// TIA Portal V18 export
// export: Created 2026-06-23T08:49:30.0253939Z, ExportSetting WithDefaults, DisplayName Totally Integrated Automation Portal, DisplayVersion V18, DisplayName TIA Portal Openness, DisplayVersion V18, DisplayName TIA Portal Version Control Interface, DisplayVersion V18, DisplayName STEP 7 Professional, DisplayVersion V18, DisplayName STEP 7 Safety, DisplayVersion V18, DisplayName WinCC Professional, DisplayVersion V18
FUNCTION "FC_Manual_Control_PLC1" : Void   // FC62, LAD
{ S7_Optimized_Access := 'TRUE' }
VERSION : 0.1
// stored: AutoNumber true, IsIECCheckEnabled false, SetENOAutomatically false, UDAEnableTagReadback false
BEGIN

REGION Network 1: Xác định trạng thái Manual Mode Active PLC1
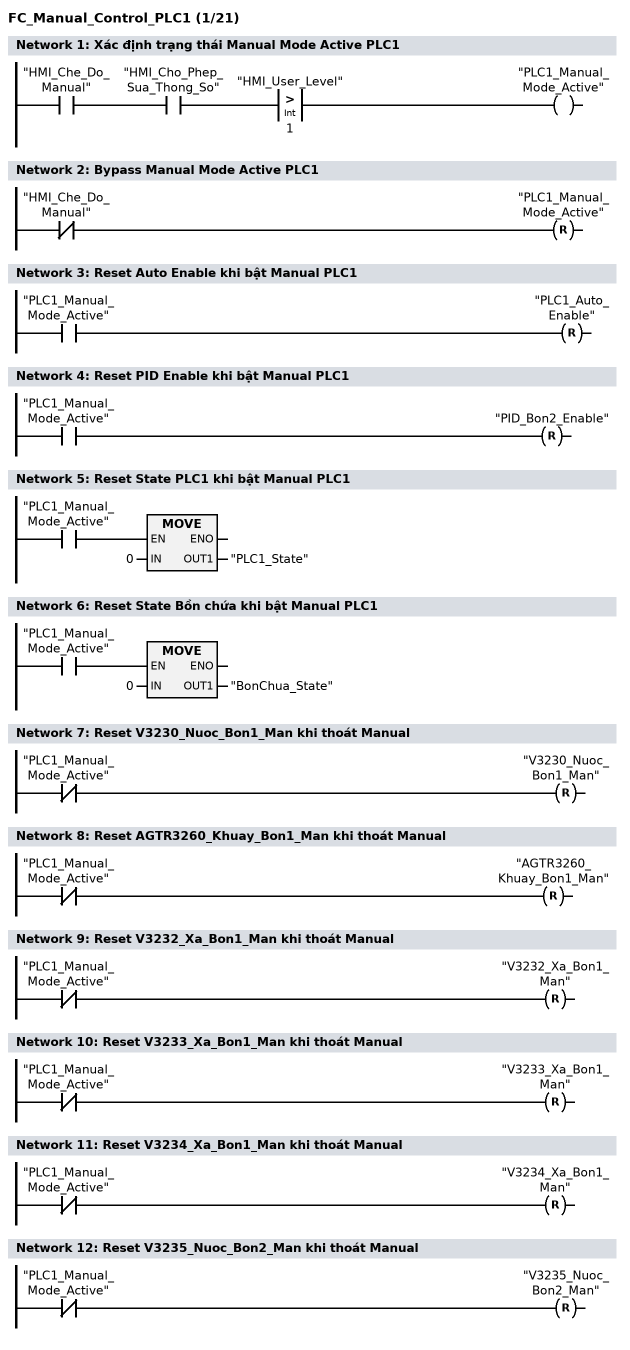
   RUNG wire#powerrail
      Contact( "HMI_Che_Do_Manual" )
      Contact( "HMI_Cho_Phep_Sua_Thong_So" )
      { S7_Templates := "SrcType := Int" } GT_Contact(in1 := "HMI_User_Level", in2 := 1)
      Coil( "PLC1_Manual_Mode_Active" )
   END_RUNG
   // the same network as SCL:
   "PLC1_Manual_Mode_Active" := "HMI_Che_Do_Manual" AND "HMI_Cho_Phep_Sua_Thong_So" AND ("HMI_User_Level" > 1);
END_REGION

REGION Network 2: Bypass Manual Mode Active PLC1
   RUNG wire#powerrail
      I_Contact( "HMI_Che_Do_Manual" )
      R_Coil( "PLC1_Manual_Mode_Active" )
   END_RUNG
   // the same network as SCL:
   IF NOT "HMI_Che_Do_Manual" THEN "PLC1_Manual_Mode_Active" := FALSE; END_IF;
END_REGION

REGION Network 3: Reset Auto Enable khi bật Manual PLC1
   RUNG wire#powerrail
      Contact( "PLC1_Manual_Mode_Active" )
      R_Coil( "PLC1_Auto_Enable" )
   END_RUNG
   // the same network as SCL:
   IF "PLC1_Manual_Mode_Active" THEN "PLC1_Auto_Enable" := FALSE; END_IF;
END_REGION

REGION Network 4: Reset PID Enable khi bật Manual PLC1
   RUNG wire#powerrail
      Contact( "PLC1_Manual_Mode_Active" )
      R_Coil( "PID_Bon2_Enable" )
   END_RUNG
   // the same network as SCL:
   IF "PLC1_Manual_Mode_Active" THEN "PID_Bon2_Enable" := FALSE; END_IF;
END_REGION

REGION Network 5: Reset State PLC1 khi bật Manual PLC1
   RUNG wire#powerrail
      Contact( "PLC1_Manual_Mode_Active" )
      { S7_GenerateENO := "TRUE" } Move(in := 0, out1 => "PLC1_State")
   END_RUNG
   // the same network as SCL:
   IF "PLC1_Manual_Mode_Active" THEN "PLC1_State" := 0; END_IF;
END_REGION

REGION Network 6: Reset State Bồn chứa khi bật Manual PLC1
   RUNG wire#powerrail
      Contact( "PLC1_Manual_Mode_Active" )
      { S7_GenerateENO := "TRUE" } Move(in := 0, out1 => "BonChua_State")
   END_RUNG
   // the same network as SCL:
   IF "PLC1_Manual_Mode_Active" THEN "BonChua_State" := 0; END_IF;
END_REGION

REGION Network 7: Reset V3230_Nuoc_Bon1_Man khi thoát Manual
   RUNG wire#powerrail
      I_Contact( "PLC1_Manual_Mode_Active" )
      R_Coil( "V3230_Nuoc_Bon1_Man" )
   END_RUNG
   // the same network as SCL:
   IF NOT "PLC1_Manual_Mode_Active" THEN "V3230_Nuoc_Bon1_Man" := FALSE; END_IF;
END_REGION

REGION Network 8: Reset AGTR3260_Khuay_Bon1_Man khi thoát Manual
   RUNG wire#powerrail
      I_Contact( "PLC1_Manual_Mode_Active" )
      R_Coil( "AGTR3260_Khuay_Bon1_Man" )
   END_RUNG
   // the same network as SCL:
   IF NOT "PLC1_Manual_Mode_Active" THEN "AGTR3260_Khuay_Bon1_Man" := FALSE; END_IF;
END_REGION

REGION Network 9: Reset V3232_Xa_Bon1_Man khi thoát Manual
   RUNG wire#powerrail
      I_Contact( "PLC1_Manual_Mode_Active" )
      R_Coil( "V3232_Xa_Bon1_Man" )
   END_RUNG
   // the same network as SCL:
   IF NOT "PLC1_Manual_Mode_Active" THEN "V3232_Xa_Bon1_Man" := FALSE; END_IF;
END_REGION

REGION Network 10: Reset V3233_Xa_Bon1_Man khi thoát Manual
   RUNG wire#powerrail
      I_Contact( "PLC1_Manual_Mode_Active" )
      R_Coil( "V3233_Xa_Bon1_Man" )
   END_RUNG
   // the same network as SCL:
   IF NOT "PLC1_Manual_Mode_Active" THEN "V3233_Xa_Bon1_Man" := FALSE; END_IF;
END_REGION

REGION Network 11: Reset V3234_Xa_Bon1_Man khi thoát Manual
   RUNG wire#powerrail
      I_Contact( "PLC1_Manual_Mode_Active" )
      R_Coil( "V3234_Xa_Bon1_Man" )
   END_RUNG
   // the same network as SCL:
   IF NOT "PLC1_Manual_Mode_Active" THEN "V3234_Xa_Bon1_Man" := FALSE; END_IF;
END_REGION

REGION Network 12: Reset V3235_Nuoc_Bon2_Man khi thoát Manual
   RUNG wire#powerrail
      I_Contact( "PLC1_Manual_Mode_Active" )
      R_Coil( "V3235_Nuoc_Bon2_Man" )
   END_RUNG
   // the same network as SCL:
   IF NOT "PLC1_Manual_Mode_Active" THEN "V3235_Nuoc_Bon2_Man" := FALSE; END_IF;
END_REGION

REGION Network 13: Reset VFD_Bon2_Run_Man khi thoát Manual
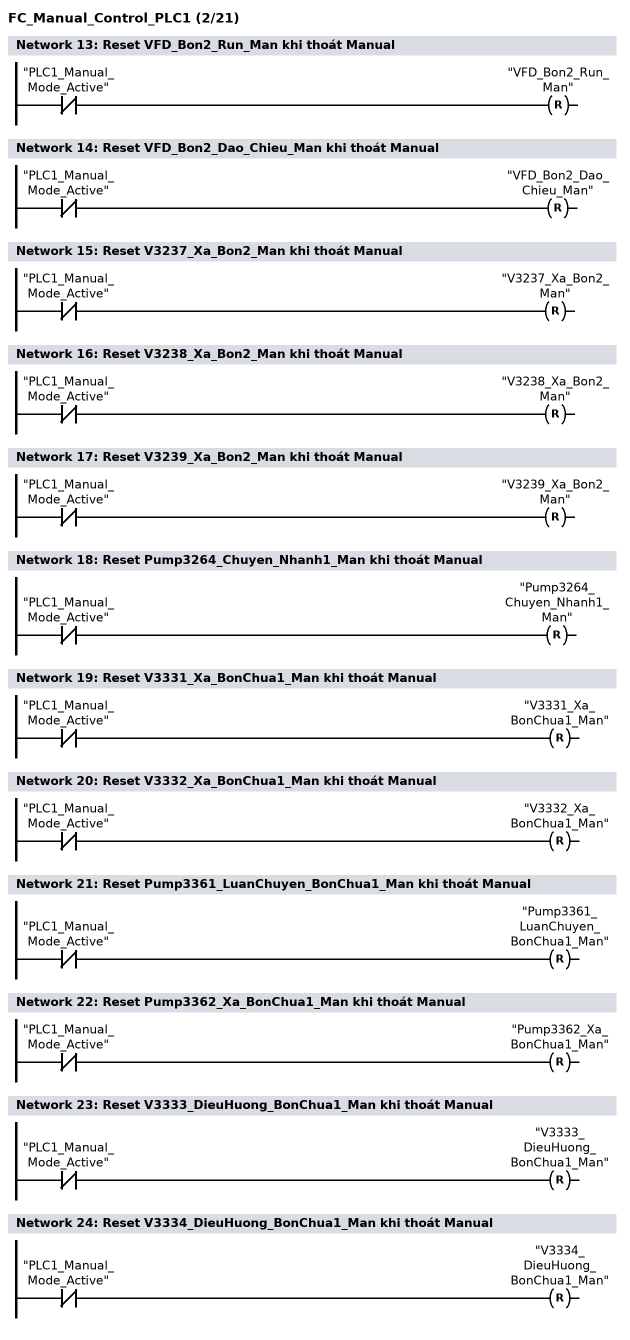
   RUNG wire#powerrail
      I_Contact( "PLC1_Manual_Mode_Active" )
      R_Coil( "VFD_Bon2_Run_Man" )
   END_RUNG
   // the same network as SCL:
   IF NOT "PLC1_Manual_Mode_Active" THEN "VFD_Bon2_Run_Man" := FALSE; END_IF;
END_REGION

REGION Network 14: Reset VFD_Bon2_Dao_Chieu_Man khi thoát Manual
   RUNG wire#powerrail
      I_Contact( "PLC1_Manual_Mode_Active" )
      R_Coil( "VFD_Bon2_Dao_Chieu_Man" )
   END_RUNG
   // the same network as SCL:
   IF NOT "PLC1_Manual_Mode_Active" THEN "VFD_Bon2_Dao_Chieu_Man" := FALSE; END_IF;
END_REGION

REGION Network 15: Reset V3237_Xa_Bon2_Man khi thoát Manual
   RUNG wire#powerrail
      I_Contact( "PLC1_Manual_Mode_Active" )
      R_Coil( "V3237_Xa_Bon2_Man" )
   END_RUNG
   // the same network as SCL:
   IF NOT "PLC1_Manual_Mode_Active" THEN "V3237_Xa_Bon2_Man" := FALSE; END_IF;
END_REGION

REGION Network 16: Reset V3238_Xa_Bon2_Man khi thoát Manual
   RUNG wire#powerrail
      I_Contact( "PLC1_Manual_Mode_Active" )
      R_Coil( "V3238_Xa_Bon2_Man" )
   END_RUNG
   // the same network as SCL:
   IF NOT "PLC1_Manual_Mode_Active" THEN "V3238_Xa_Bon2_Man" := FALSE; END_IF;
END_REGION

REGION Network 17: Reset V3239_Xa_Bon2_Man khi thoát Manual
   RUNG wire#powerrail
      I_Contact( "PLC1_Manual_Mode_Active" )
      R_Coil( "V3239_Xa_Bon2_Man" )
   END_RUNG
   // the same network as SCL:
   IF NOT "PLC1_Manual_Mode_Active" THEN "V3239_Xa_Bon2_Man" := FALSE; END_IF;
END_REGION

REGION Network 18: Reset Pump3264_Chuyen_Nhanh1_Man khi thoát Manual
   RUNG wire#powerrail
      I_Contact( "PLC1_Manual_Mode_Active" )
      R_Coil( "Pump3264_Chuyen_Nhanh1_Man" )
   END_RUNG
   // the same network as SCL:
   IF NOT "PLC1_Manual_Mode_Active" THEN "Pump3264_Chuyen_Nhanh1_Man" := FALSE; END_IF;
END_REGION

REGION Network 19: Reset V3331_Xa_BonChua1_Man khi thoát Manual
   RUNG wire#powerrail
      I_Contact( "PLC1_Manual_Mode_Active" )
      R_Coil( "V3331_Xa_BonChua1_Man" )
   END_RUNG
   // the same network as SCL:
   IF NOT "PLC1_Manual_Mode_Active" THEN "V3331_Xa_BonChua1_Man" := FALSE; END_IF;
END_REGION

REGION Network 20: Reset V3332_Xa_BonChua1_Man khi thoát Manual
   RUNG wire#powerrail
      I_Contact( "PLC1_Manual_Mode_Active" )
      R_Coil( "V3332_Xa_BonChua1_Man" )
   END_RUNG
   // the same network as SCL:
   IF NOT "PLC1_Manual_Mode_Active" THEN "V3332_Xa_BonChua1_Man" := FALSE; END_IF;
END_REGION

REGION Network 21: Reset Pump3361_LuanChuyen_BonChua1_Man khi thoát Manual
   RUNG wire#powerrail
      I_Contact( "PLC1_Manual_Mode_Active" )
      R_Coil( "Pump3361_LuanChuyen_BonChua1_Man" )
   END_RUNG
   // the same network as SCL:
   IF NOT "PLC1_Manual_Mode_Active" THEN "Pump3361_LuanChuyen_BonChua1_Man" := FALSE; END_IF;
END_REGION

REGION Network 22: Reset Pump3362_Xa_BonChua1_Man khi thoát Manual
   RUNG wire#powerrail
      I_Contact( "PLC1_Manual_Mode_Active" )
      R_Coil( "Pump3362_Xa_BonChua1_Man" )
   END_RUNG
   // the same network as SCL:
   IF NOT "PLC1_Manual_Mode_Active" THEN "Pump3362_Xa_BonChua1_Man" := FALSE; END_IF;
END_REGION

REGION Network 23: Reset V3333_DieuHuong_BonChua1_Man khi thoát Manual
   RUNG wire#powerrail
      I_Contact( "PLC1_Manual_Mode_Active" )
      R_Coil( "V3333_DieuHuong_BonChua1_Man" )
   END_RUNG
   // the same network as SCL:
   IF NOT "PLC1_Manual_Mode_Active" THEN "V3333_DieuHuong_BonChua1_Man" := FALSE; END_IF;
END_REGION

REGION Network 24: Reset V3334_DieuHuong_BonChua1_Man khi thoát Manual
   RUNG wire#powerrail
      I_Contact( "PLC1_Manual_Mode_Active" )
      R_Coil( "V3334_DieuHuong_BonChua1_Man" )
   END_RUNG
   // the same network as SCL:
   IF NOT "PLC1_Manual_Mode_Active" THEN "V3334_DieuHuong_BonChua1_Man" := FALSE; END_IF;
END_REGION

REGION Network 25: Reset V3335_DieuHuong_BonChua1_Man khi thoát Manual
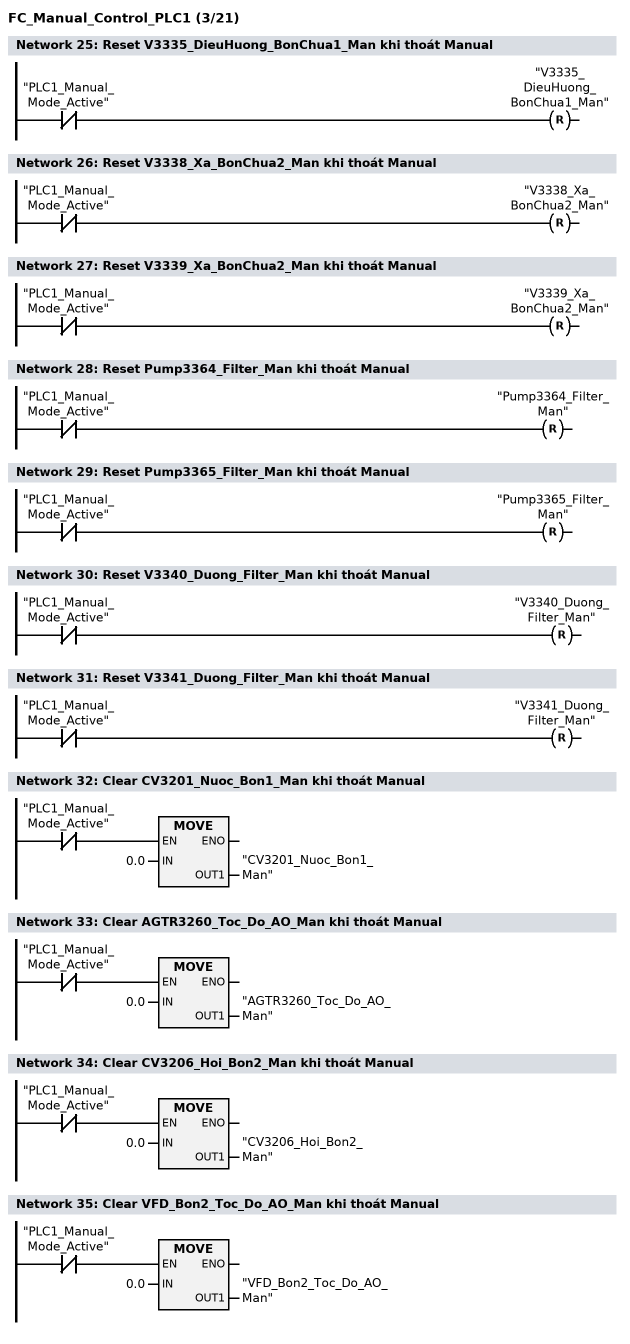
   RUNG wire#powerrail
      I_Contact( "PLC1_Manual_Mode_Active" )
      R_Coil( "V3335_DieuHuong_BonChua1_Man" )
   END_RUNG
   // the same network as SCL:
   IF NOT "PLC1_Manual_Mode_Active" THEN "V3335_DieuHuong_BonChua1_Man" := FALSE; END_IF;
END_REGION

REGION Network 26: Reset V3338_Xa_BonChua2_Man khi thoát Manual
   RUNG wire#powerrail
      I_Contact( "PLC1_Manual_Mode_Active" )
      R_Coil( "V3338_Xa_BonChua2_Man" )
   END_RUNG
   // the same network as SCL:
   IF NOT "PLC1_Manual_Mode_Active" THEN "V3338_Xa_BonChua2_Man" := FALSE; END_IF;
END_REGION

REGION Network 27: Reset V3339_Xa_BonChua2_Man khi thoát Manual
   RUNG wire#powerrail
      I_Contact( "PLC1_Manual_Mode_Active" )
      R_Coil( "V3339_Xa_BonChua2_Man" )
   END_RUNG
   // the same network as SCL:
   IF NOT "PLC1_Manual_Mode_Active" THEN "V3339_Xa_BonChua2_Man" := FALSE; END_IF;
END_REGION

REGION Network 28: Reset Pump3364_Filter_Man khi thoát Manual
   RUNG wire#powerrail
      I_Contact( "PLC1_Manual_Mode_Active" )
      R_Coil( "Pump3364_Filter_Man" )
   END_RUNG
   // the same network as SCL:
   IF NOT "PLC1_Manual_Mode_Active" THEN "Pump3364_Filter_Man" := FALSE; END_IF;
END_REGION

REGION Network 29: Reset Pump3365_Filter_Man khi thoát Manual
   RUNG wire#powerrail
      I_Contact( "PLC1_Manual_Mode_Active" )
      R_Coil( "Pump3365_Filter_Man" )
   END_RUNG
   // the same network as SCL:
   IF NOT "PLC1_Manual_Mode_Active" THEN "Pump3365_Filter_Man" := FALSE; END_IF;
END_REGION

REGION Network 30: Reset V3340_Duong_Filter_Man khi thoát Manual
   RUNG wire#powerrail
      I_Contact( "PLC1_Manual_Mode_Active" )
      R_Coil( "V3340_Duong_Filter_Man" )
   END_RUNG
   // the same network as SCL:
   IF NOT "PLC1_Manual_Mode_Active" THEN "V3340_Duong_Filter_Man" := FALSE; END_IF;
END_REGION

REGION Network 31: Reset V3341_Duong_Filter_Man khi thoát Manual
   RUNG wire#powerrail
      I_Contact( "PLC1_Manual_Mode_Active" )
      R_Coil( "V3341_Duong_Filter_Man" )
   END_RUNG
   // the same network as SCL:
   IF NOT "PLC1_Manual_Mode_Active" THEN "V3341_Duong_Filter_Man" := FALSE; END_IF;
END_REGION

REGION Network 32: Clear CV3201_Nuoc_Bon1_Man khi thoát Manual
   RUNG wire#powerrail
      I_Contact( "PLC1_Manual_Mode_Active" )
      { S7_GenerateENO := "TRUE" } Move(in := 0.0, out1 => "CV3201_Nuoc_Bon1_Man")
   END_RUNG
   // the same network as SCL:
   IF NOT "PLC1_Manual_Mode_Active" THEN "CV3201_Nuoc_Bon1_Man" := 0.0; END_IF;
END_REGION

REGION Network 33: Clear AGTR3260_Toc_Do_AO_Man khi thoát Manual
   RUNG wire#powerrail
      I_Contact( "PLC1_Manual_Mode_Active" )
      { S7_GenerateENO := "TRUE" } Move(in := 0.0, out1 => "AGTR3260_Toc_Do_AO_Man")
   END_RUNG
   // the same network as SCL:
   IF NOT "PLC1_Manual_Mode_Active" THEN "AGTR3260_Toc_Do_AO_Man" := 0.0; END_IF;
END_REGION

REGION Network 34: Clear CV3206_Hoi_Bon2_Man khi thoát Manual
   RUNG wire#powerrail
      I_Contact( "PLC1_Manual_Mode_Active" )
      { S7_GenerateENO := "TRUE" } Move(in := 0.0, out1 => "CV3206_Hoi_Bon2_Man")
   END_RUNG
   // the same network as SCL:
   IF NOT "PLC1_Manual_Mode_Active" THEN "CV3206_Hoi_Bon2_Man" := 0.0; END_IF;
END_REGION

REGION Network 35: Clear VFD_Bon2_Toc_Do_AO_Man khi thoát Manual
   RUNG wire#powerrail
      I_Contact( "PLC1_Manual_Mode_Active" )
      { S7_GenerateENO := "TRUE" } Move(in := 0.0, out1 => "VFD_Bon2_Toc_Do_AO_Man")
   END_RUNG
   // the same network as SCL:
   IF NOT "PLC1_Manual_Mode_Active" THEN "VFD_Bon2_Toc_Do_AO_Man" := 0.0; END_IF;
END_REGION

REGION Network 36: Clear CV3304_Nuoc_Lam_Mat_Man khi thoát Manual
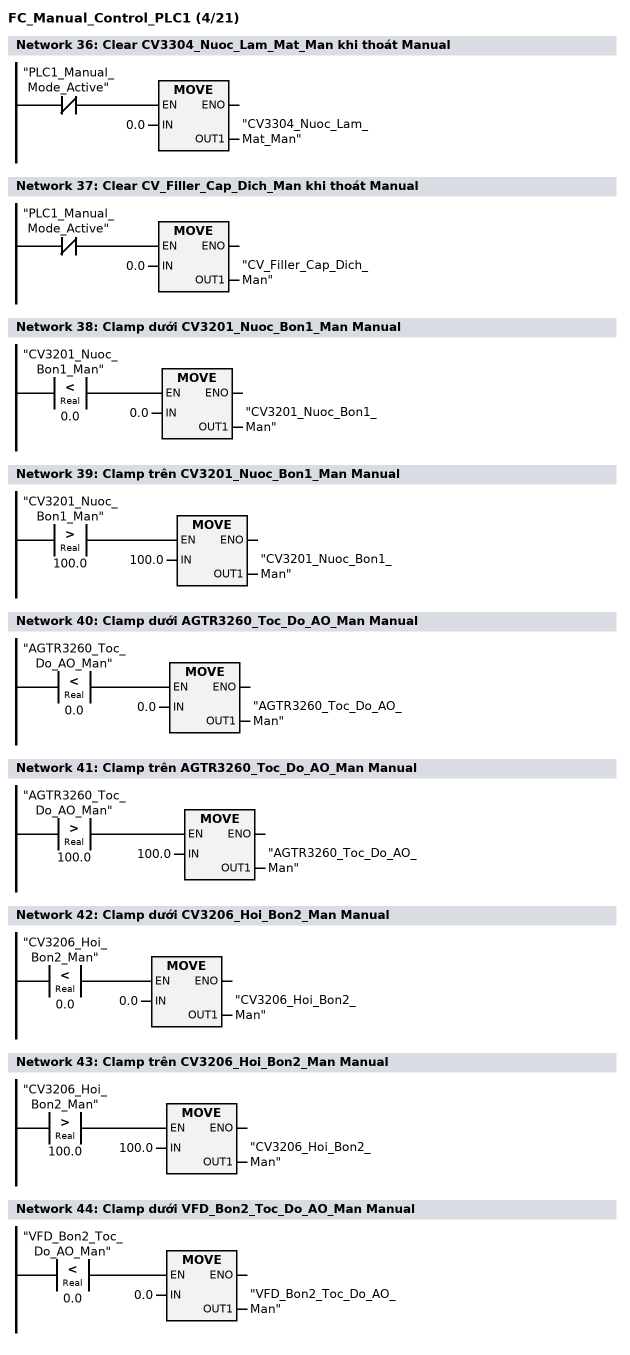
   RUNG wire#powerrail
      I_Contact( "PLC1_Manual_Mode_Active" )
      { S7_GenerateENO := "TRUE" } Move(in := 0.0, out1 => "CV3304_Nuoc_Lam_Mat_Man")
   END_RUNG
   // the same network as SCL:
   IF NOT "PLC1_Manual_Mode_Active" THEN "CV3304_Nuoc_Lam_Mat_Man" := 0.0; END_IF;
END_REGION

REGION Network 37: Clear CV_Filler_Cap_Dich_Man khi thoát Manual
   RUNG wire#powerrail
      I_Contact( "PLC1_Manual_Mode_Active" )
      { S7_GenerateENO := "TRUE" } Move(in := 0.0, out1 => "CV_Filler_Cap_Dich_Man")
   END_RUNG
   // the same network as SCL:
   IF NOT "PLC1_Manual_Mode_Active" THEN "CV_Filler_Cap_Dich_Man" := 0.0; END_IF;
END_REGION

REGION Network 38: Clamp dưới CV3201_Nuoc_Bon1_Man Manual
   RUNG wire#powerrail
      { S7_Templates := "SrcType := Real" } LT_Contact(in1 := "CV3201_Nuoc_Bon1_Man", in2 := 0.0)
      { S7_GenerateENO := "TRUE" } Move(in := 0.0, out1 => "CV3201_Nuoc_Bon1_Man")
   END_RUNG
   // the same network as SCL:
   IF "CV3201_Nuoc_Bon1_Man" < 0.0 THEN "CV3201_Nuoc_Bon1_Man" := 0.0; END_IF;
END_REGION

REGION Network 39: Clamp trên CV3201_Nuoc_Bon1_Man Manual
   RUNG wire#powerrail
      { S7_Templates := "SrcType := Real" } GT_Contact(in1 := "CV3201_Nuoc_Bon1_Man", in2 := 100.0)
      { S7_GenerateENO := "TRUE" } Move(in := 100.0, out1 => "CV3201_Nuoc_Bon1_Man")
   END_RUNG
   // the same network as SCL:
   IF "CV3201_Nuoc_Bon1_Man" > 100.0 THEN "CV3201_Nuoc_Bon1_Man" := 100.0; END_IF;
END_REGION

REGION Network 40: Clamp dưới AGTR3260_Toc_Do_AO_Man Manual
   RUNG wire#powerrail
      { S7_Templates := "SrcType := Real" } LT_Contact(in1 := "AGTR3260_Toc_Do_AO_Man", in2 := 0.0)
      { S7_GenerateENO := "TRUE" } Move(in := 0.0, out1 => "AGTR3260_Toc_Do_AO_Man")
   END_RUNG
   // the same network as SCL:
   IF "AGTR3260_Toc_Do_AO_Man" < 0.0 THEN "AGTR3260_Toc_Do_AO_Man" := 0.0; END_IF;
END_REGION

REGION Network 41: Clamp trên AGTR3260_Toc_Do_AO_Man Manual
   RUNG wire#powerrail
      { S7_Templates := "SrcType := Real" } GT_Contact(in1 := "AGTR3260_Toc_Do_AO_Man", in2 := 100.0)
      { S7_GenerateENO := "TRUE" } Move(in := 100.0, out1 => "AGTR3260_Toc_Do_AO_Man")
   END_RUNG
   // the same network as SCL:
   IF "AGTR3260_Toc_Do_AO_Man" > 100.0 THEN "AGTR3260_Toc_Do_AO_Man" := 100.0; END_IF;
END_REGION

REGION Network 42: Clamp dưới CV3206_Hoi_Bon2_Man Manual
   RUNG wire#powerrail
      { S7_Templates := "SrcType := Real" } LT_Contact(in1 := "CV3206_Hoi_Bon2_Man", in2 := 0.0)
      { S7_GenerateENO := "TRUE" } Move(in := 0.0, out1 => "CV3206_Hoi_Bon2_Man")
   END_RUNG
   // the same network as SCL:
   IF "CV3206_Hoi_Bon2_Man" < 0.0 THEN "CV3206_Hoi_Bon2_Man" := 0.0; END_IF;
END_REGION

REGION Network 43: Clamp trên CV3206_Hoi_Bon2_Man Manual
   RUNG wire#powerrail
      { S7_Templates := "SrcType := Real" } GT_Contact(in1 := "CV3206_Hoi_Bon2_Man", in2 := 100.0)
      { S7_GenerateENO := "TRUE" } Move(in := 100.0, out1 => "CV3206_Hoi_Bon2_Man")
   END_RUNG
   // the same network as SCL:
   IF "CV3206_Hoi_Bon2_Man" > 100.0 THEN "CV3206_Hoi_Bon2_Man" := 100.0; END_IF;
END_REGION

REGION Network 44: Clamp dưới VFD_Bon2_Toc_Do_AO_Man Manual
   RUNG wire#powerrail
      { S7_Templates := "SrcType := Real" } LT_Contact(in1 := "VFD_Bon2_Toc_Do_AO_Man", in2 := 0.0)
      { S7_GenerateENO := "TRUE" } Move(in := 0.0, out1 => "VFD_Bon2_Toc_Do_AO_Man")
   END_RUNG
   // the same network as SCL:
   IF "VFD_Bon2_Toc_Do_AO_Man" < 0.0 THEN "VFD_Bon2_Toc_Do_AO_Man" := 0.0; END_IF;
END_REGION

REGION Network 45: Clamp trên VFD_Bon2_Toc_Do_AO_Man Manual
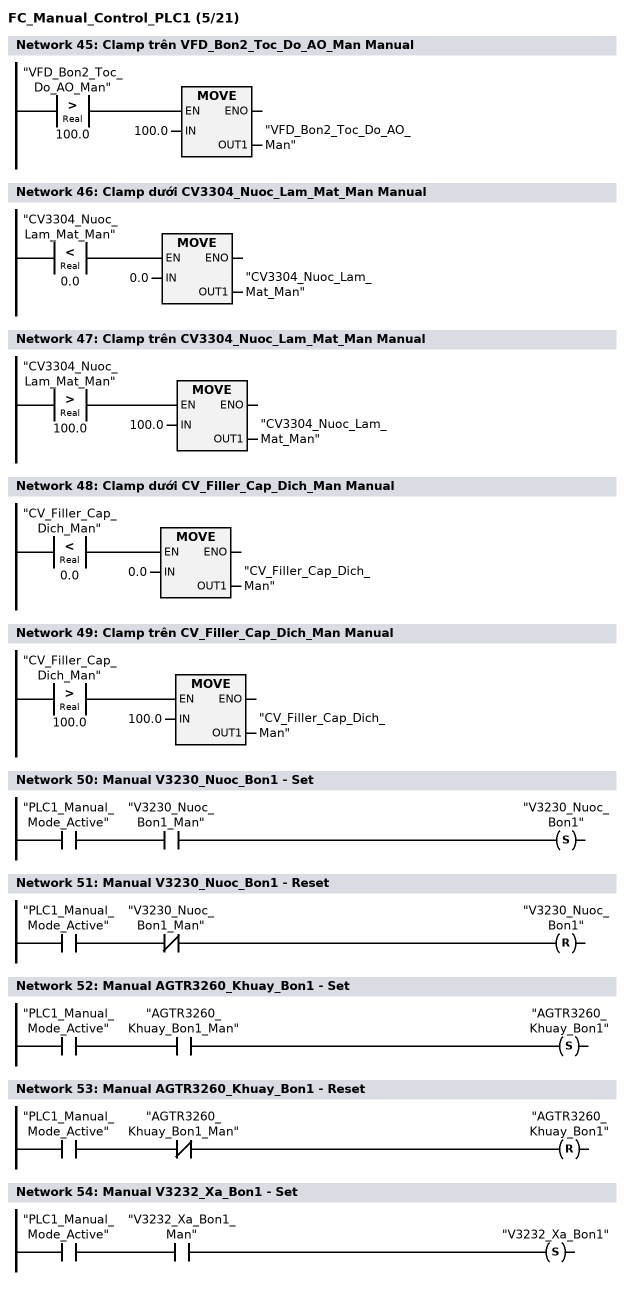
   RUNG wire#powerrail
      { S7_Templates := "SrcType := Real" } GT_Contact(in1 := "VFD_Bon2_Toc_Do_AO_Man", in2 := 100.0)
      { S7_GenerateENO := "TRUE" } Move(in := 100.0, out1 => "VFD_Bon2_Toc_Do_AO_Man")
   END_RUNG
   // the same network as SCL:
   IF "VFD_Bon2_Toc_Do_AO_Man" > 100.0 THEN "VFD_Bon2_Toc_Do_AO_Man" := 100.0; END_IF;
END_REGION

REGION Network 46: Clamp dưới CV3304_Nuoc_Lam_Mat_Man Manual
   RUNG wire#powerrail
      { S7_Templates := "SrcType := Real" } LT_Contact(in1 := "CV3304_Nuoc_Lam_Mat_Man", in2 := 0.0)
      { S7_GenerateENO := "TRUE" } Move(in := 0.0, out1 => "CV3304_Nuoc_Lam_Mat_Man")
   END_RUNG
   // the same network as SCL:
   IF "CV3304_Nuoc_Lam_Mat_Man" < 0.0 THEN "CV3304_Nuoc_Lam_Mat_Man" := 0.0; END_IF;
END_REGION

REGION Network 47: Clamp trên CV3304_Nuoc_Lam_Mat_Man Manual
   RUNG wire#powerrail
      { S7_Templates := "SrcType := Real" } GT_Contact(in1 := "CV3304_Nuoc_Lam_Mat_Man", in2 := 100.0)
      { S7_GenerateENO := "TRUE" } Move(in := 100.0, out1 => "CV3304_Nuoc_Lam_Mat_Man")
   END_RUNG
   // the same network as SCL:
   IF "CV3304_Nuoc_Lam_Mat_Man" > 100.0 THEN "CV3304_Nuoc_Lam_Mat_Man" := 100.0; END_IF;
END_REGION

REGION Network 48: Clamp dưới CV_Filler_Cap_Dich_Man Manual
   RUNG wire#powerrail
      { S7_Templates := "SrcType := Real" } LT_Contact(in1 := "CV_Filler_Cap_Dich_Man", in2 := 0.0)
      { S7_GenerateENO := "TRUE" } Move(in := 0.0, out1 => "CV_Filler_Cap_Dich_Man")
   END_RUNG
   // the same network as SCL:
   IF "CV_Filler_Cap_Dich_Man" < 0.0 THEN "CV_Filler_Cap_Dich_Man" := 0.0; END_IF;
END_REGION

REGION Network 49: Clamp trên CV_Filler_Cap_Dich_Man Manual
   RUNG wire#powerrail
      { S7_Templates := "SrcType := Real" } GT_Contact(in1 := "CV_Filler_Cap_Dich_Man", in2 := 100.0)
      { S7_GenerateENO := "TRUE" } Move(in := 100.0, out1 => "CV_Filler_Cap_Dich_Man")
   END_RUNG
   // the same network as SCL:
   IF "CV_Filler_Cap_Dich_Man" > 100.0 THEN "CV_Filler_Cap_Dich_Man" := 100.0; END_IF;
END_REGION

REGION Network 50: Manual V3230_Nuoc_Bon1 - Set
   RUNG wire#powerrail
      Contact( "PLC1_Manual_Mode_Active" )
      Contact( "V3230_Nuoc_Bon1_Man" )
      S_Coil( "V3230_Nuoc_Bon1" )
   END_RUNG
   // the same network as SCL:
   IF "PLC1_Manual_Mode_Active" AND "V3230_Nuoc_Bon1_Man" THEN "V3230_Nuoc_Bon1" := TRUE; END_IF;
END_REGION

REGION Network 51: Manual V3230_Nuoc_Bon1 - Reset
   RUNG wire#powerrail
      Contact( "PLC1_Manual_Mode_Active" )
      I_Contact( "V3230_Nuoc_Bon1_Man" )
      R_Coil( "V3230_Nuoc_Bon1" )
   END_RUNG
   // the same network as SCL:
   IF "PLC1_Manual_Mode_Active" AND NOT "V3230_Nuoc_Bon1_Man" THEN "V3230_Nuoc_Bon1" := FALSE; END_IF;
END_REGION

REGION Network 52: Manual AGTR3260_Khuay_Bon1 - Set
   RUNG wire#powerrail
      Contact( "PLC1_Manual_Mode_Active" )
      Contact( "AGTR3260_Khuay_Bon1_Man" )
      S_Coil( "AGTR3260_Khuay_Bon1" )
   END_RUNG
   // the same network as SCL:
   IF "PLC1_Manual_Mode_Active" AND "AGTR3260_Khuay_Bon1_Man" THEN "AGTR3260_Khuay_Bon1" := TRUE; END_IF;
END_REGION

REGION Network 53: Manual AGTR3260_Khuay_Bon1 - Reset
   RUNG wire#powerrail
      Contact( "PLC1_Manual_Mode_Active" )
      I_Contact( "AGTR3260_Khuay_Bon1_Man" )
      R_Coil( "AGTR3260_Khuay_Bon1" )
   END_RUNG
   // the same network as SCL:
   IF "PLC1_Manual_Mode_Active" AND NOT "AGTR3260_Khuay_Bon1_Man" THEN
       "AGTR3260_Khuay_Bon1" := FALSE;
   END_IF;
END_REGION

REGION Network 54: Manual V3232_Xa_Bon1 - Set
   RUNG wire#powerrail
      Contact( "PLC1_Manual_Mode_Active" )
      Contact( "V3232_Xa_Bon1_Man" )
      S_Coil( "V3232_Xa_Bon1" )
   END_RUNG
   // the same network as SCL:
   IF "PLC1_Manual_Mode_Active" AND "V3232_Xa_Bon1_Man" THEN "V3232_Xa_Bon1" := TRUE; END_IF;
END_REGION

REGION Network 55: Manual V3232_Xa_Bon1 - Reset
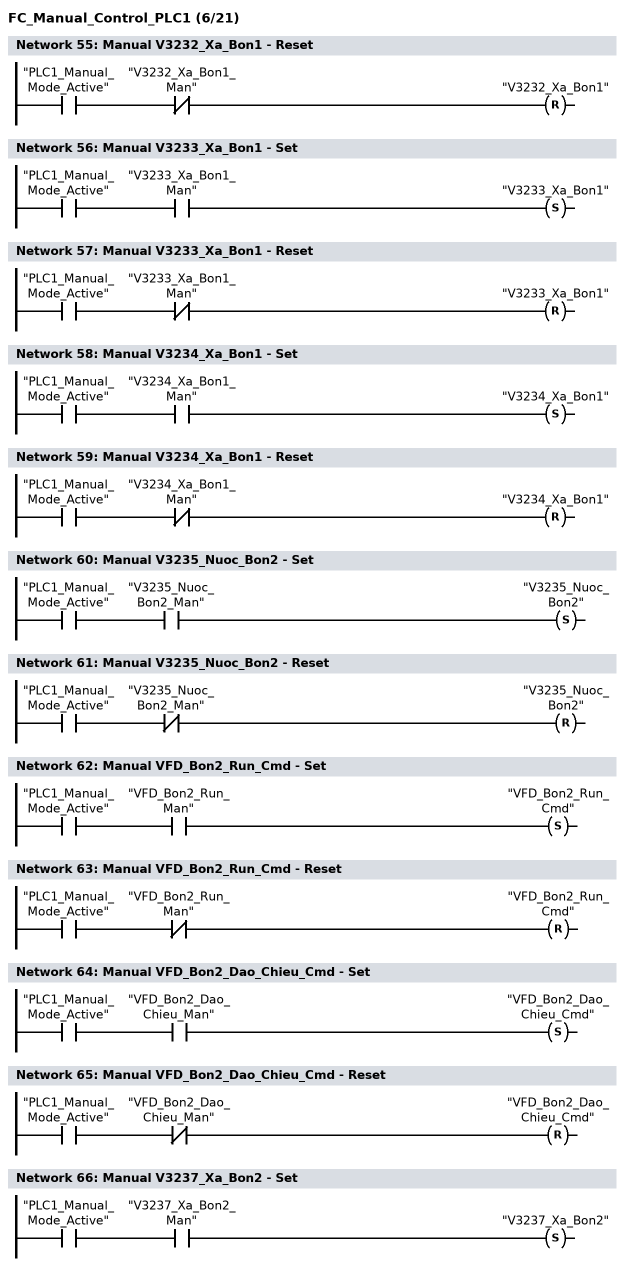
   RUNG wire#powerrail
      Contact( "PLC1_Manual_Mode_Active" )
      I_Contact( "V3232_Xa_Bon1_Man" )
      R_Coil( "V3232_Xa_Bon1" )
   END_RUNG
   // the same network as SCL:
   IF "PLC1_Manual_Mode_Active" AND NOT "V3232_Xa_Bon1_Man" THEN "V3232_Xa_Bon1" := FALSE; END_IF;
END_REGION

REGION Network 56: Manual V3233_Xa_Bon1 - Set
   RUNG wire#powerrail
      Contact( "PLC1_Manual_Mode_Active" )
      Contact( "V3233_Xa_Bon1_Man" )
      S_Coil( "V3233_Xa_Bon1" )
   END_RUNG
   // the same network as SCL:
   IF "PLC1_Manual_Mode_Active" AND "V3233_Xa_Bon1_Man" THEN "V3233_Xa_Bon1" := TRUE; END_IF;
END_REGION

REGION Network 57: Manual V3233_Xa_Bon1 - Reset
   RUNG wire#powerrail
      Contact( "PLC1_Manual_Mode_Active" )
      I_Contact( "V3233_Xa_Bon1_Man" )
      R_Coil( "V3233_Xa_Bon1" )
   END_RUNG
   // the same network as SCL:
   IF "PLC1_Manual_Mode_Active" AND NOT "V3233_Xa_Bon1_Man" THEN "V3233_Xa_Bon1" := FALSE; END_IF;
END_REGION

REGION Network 58: Manual V3234_Xa_Bon1 - Set
   RUNG wire#powerrail
      Contact( "PLC1_Manual_Mode_Active" )
      Contact( "V3234_Xa_Bon1_Man" )
      S_Coil( "V3234_Xa_Bon1" )
   END_RUNG
   // the same network as SCL:
   IF "PLC1_Manual_Mode_Active" AND "V3234_Xa_Bon1_Man" THEN "V3234_Xa_Bon1" := TRUE; END_IF;
END_REGION

REGION Network 59: Manual V3234_Xa_Bon1 - Reset
   RUNG wire#powerrail
      Contact( "PLC1_Manual_Mode_Active" )
      I_Contact( "V3234_Xa_Bon1_Man" )
      R_Coil( "V3234_Xa_Bon1" )
   END_RUNG
   // the same network as SCL:
   IF "PLC1_Manual_Mode_Active" AND NOT "V3234_Xa_Bon1_Man" THEN "V3234_Xa_Bon1" := FALSE; END_IF;
END_REGION

REGION Network 60: Manual V3235_Nuoc_Bon2 - Set
   RUNG wire#powerrail
      Contact( "PLC1_Manual_Mode_Active" )
      Contact( "V3235_Nuoc_Bon2_Man" )
      S_Coil( "V3235_Nuoc_Bon2" )
   END_RUNG
   // the same network as SCL:
   IF "PLC1_Manual_Mode_Active" AND "V3235_Nuoc_Bon2_Man" THEN "V3235_Nuoc_Bon2" := TRUE; END_IF;
END_REGION

REGION Network 61: Manual V3235_Nuoc_Bon2 - Reset
   RUNG wire#powerrail
      Contact( "PLC1_Manual_Mode_Active" )
      I_Contact( "V3235_Nuoc_Bon2_Man" )
      R_Coil( "V3235_Nuoc_Bon2" )
   END_RUNG
   // the same network as SCL:
   IF "PLC1_Manual_Mode_Active" AND NOT "V3235_Nuoc_Bon2_Man" THEN "V3235_Nuoc_Bon2" := FALSE; END_IF;
END_REGION

REGION Network 62: Manual VFD_Bon2_Run_Cmd - Set
   RUNG wire#powerrail
      Contact( "PLC1_Manual_Mode_Active" )
      Contact( "VFD_Bon2_Run_Man" )
      S_Coil( "VFD_Bon2_Run_Cmd" )
   END_RUNG
   // the same network as SCL:
   IF "PLC1_Manual_Mode_Active" AND "VFD_Bon2_Run_Man" THEN "VFD_Bon2_Run_Cmd" := TRUE; END_IF;
END_REGION

REGION Network 63: Manual VFD_Bon2_Run_Cmd - Reset
   RUNG wire#powerrail
      Contact( "PLC1_Manual_Mode_Active" )
      I_Contact( "VFD_Bon2_Run_Man" )
      R_Coil( "VFD_Bon2_Run_Cmd" )
   END_RUNG
   // the same network as SCL:
   IF "PLC1_Manual_Mode_Active" AND NOT "VFD_Bon2_Run_Man" THEN "VFD_Bon2_Run_Cmd" := FALSE; END_IF;
END_REGION

REGION Network 64: Manual VFD_Bon2_Dao_Chieu_Cmd - Set
   RUNG wire#powerrail
      Contact( "PLC1_Manual_Mode_Active" )
      Contact( "VFD_Bon2_Dao_Chieu_Man" )
      S_Coil( "VFD_Bon2_Dao_Chieu_Cmd" )
   END_RUNG
   // the same network as SCL:
   IF "PLC1_Manual_Mode_Active" AND "VFD_Bon2_Dao_Chieu_Man" THEN "VFD_Bon2_Dao_Chieu_Cmd" := TRUE; END_IF;
END_REGION

REGION Network 65: Manual VFD_Bon2_Dao_Chieu_Cmd - Reset
   RUNG wire#powerrail
      Contact( "PLC1_Manual_Mode_Active" )
      I_Contact( "VFD_Bon2_Dao_Chieu_Man" )
      R_Coil( "VFD_Bon2_Dao_Chieu_Cmd" )
   END_RUNG
   // the same network as SCL:
   IF "PLC1_Manual_Mode_Active" AND NOT "VFD_Bon2_Dao_Chieu_Man" THEN
       "VFD_Bon2_Dao_Chieu_Cmd" := FALSE;
   END_IF;
END_REGION

REGION Network 66: Manual V3237_Xa_Bon2 - Set
   RUNG wire#powerrail
      Contact( "PLC1_Manual_Mode_Active" )
      Contact( "V3237_Xa_Bon2_Man" )
      S_Coil( "V3237_Xa_Bon2" )
   END_RUNG
   // the same network as SCL:
   IF "PLC1_Manual_Mode_Active" AND "V3237_Xa_Bon2_Man" THEN "V3237_Xa_Bon2" := TRUE; END_IF;
END_REGION

REGION Network 67: Manual V3237_Xa_Bon2 - Reset
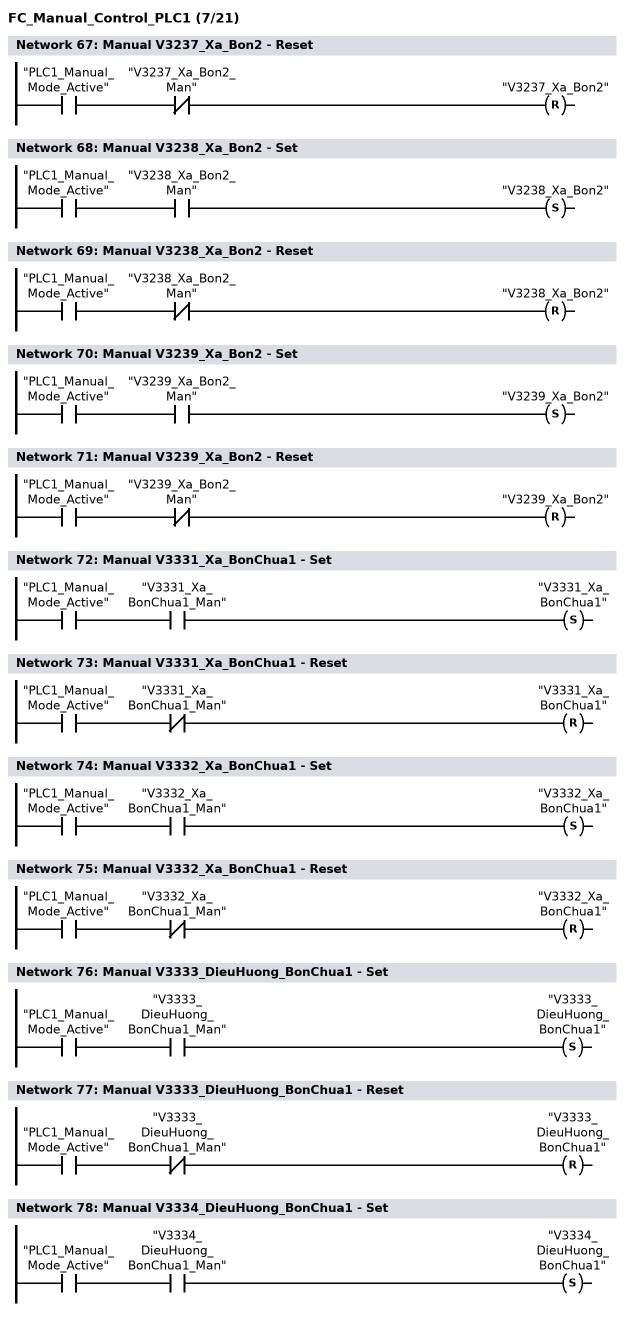
   RUNG wire#powerrail
      Contact( "PLC1_Manual_Mode_Active" )
      I_Contact( "V3237_Xa_Bon2_Man" )
      R_Coil( "V3237_Xa_Bon2" )
   END_RUNG
   // the same network as SCL:
   IF "PLC1_Manual_Mode_Active" AND NOT "V3237_Xa_Bon2_Man" THEN "V3237_Xa_Bon2" := FALSE; END_IF;
END_REGION

REGION Network 68: Manual V3238_Xa_Bon2 - Set
   RUNG wire#powerrail
      Contact( "PLC1_Manual_Mode_Active" )
      Contact( "V3238_Xa_Bon2_Man" )
      S_Coil( "V3238_Xa_Bon2" )
   END_RUNG
   // the same network as SCL:
   IF "PLC1_Manual_Mode_Active" AND "V3238_Xa_Bon2_Man" THEN "V3238_Xa_Bon2" := TRUE; END_IF;
END_REGION

REGION Network 69: Manual V3238_Xa_Bon2 - Reset
   RUNG wire#powerrail
      Contact( "PLC1_Manual_Mode_Active" )
      I_Contact( "V3238_Xa_Bon2_Man" )
      R_Coil( "V3238_Xa_Bon2" )
   END_RUNG
   // the same network as SCL:
   IF "PLC1_Manual_Mode_Active" AND NOT "V3238_Xa_Bon2_Man" THEN "V3238_Xa_Bon2" := FALSE; END_IF;
END_REGION

REGION Network 70: Manual V3239_Xa_Bon2 - Set
   RUNG wire#powerrail
      Contact( "PLC1_Manual_Mode_Active" )
      Contact( "V3239_Xa_Bon2_Man" )
      S_Coil( "V3239_Xa_Bon2" )
   END_RUNG
   // the same network as SCL:
   IF "PLC1_Manual_Mode_Active" AND "V3239_Xa_Bon2_Man" THEN "V3239_Xa_Bon2" := TRUE; END_IF;
END_REGION

REGION Network 71: Manual V3239_Xa_Bon2 - Reset
   RUNG wire#powerrail
      Contact( "PLC1_Manual_Mode_Active" )
      I_Contact( "V3239_Xa_Bon2_Man" )
      R_Coil( "V3239_Xa_Bon2" )
   END_RUNG
   // the same network as SCL:
   IF "PLC1_Manual_Mode_Active" AND NOT "V3239_Xa_Bon2_Man" THEN "V3239_Xa_Bon2" := FALSE; END_IF;
END_REGION

REGION Network 72: Manual V3331_Xa_BonChua1 - Set
   RUNG wire#powerrail
      Contact( "PLC1_Manual_Mode_Active" )
      Contact( "V3331_Xa_BonChua1_Man" )
      S_Coil( "V3331_Xa_BonChua1" )
   END_RUNG
   // the same network as SCL:
   IF "PLC1_Manual_Mode_Active" AND "V3331_Xa_BonChua1_Man" THEN "V3331_Xa_BonChua1" := TRUE; END_IF;
END_REGION

REGION Network 73: Manual V3331_Xa_BonChua1 - Reset
   RUNG wire#powerrail
      Contact( "PLC1_Manual_Mode_Active" )
      I_Contact( "V3331_Xa_BonChua1_Man" )
      R_Coil( "V3331_Xa_BonChua1" )
   END_RUNG
   // the same network as SCL:
   IF "PLC1_Manual_Mode_Active" AND NOT "V3331_Xa_BonChua1_Man" THEN "V3331_Xa_BonChua1" := FALSE; END_IF;
END_REGION

REGION Network 74: Manual V3332_Xa_BonChua1 - Set
   RUNG wire#powerrail
      Contact( "PLC1_Manual_Mode_Active" )
      Contact( "V3332_Xa_BonChua1_Man" )
      S_Coil( "V3332_Xa_BonChua1" )
   END_RUNG
   // the same network as SCL:
   IF "PLC1_Manual_Mode_Active" AND "V3332_Xa_BonChua1_Man" THEN "V3332_Xa_BonChua1" := TRUE; END_IF;
END_REGION

REGION Network 75: Manual V3332_Xa_BonChua1 - Reset
   RUNG wire#powerrail
      Contact( "PLC1_Manual_Mode_Active" )
      I_Contact( "V3332_Xa_BonChua1_Man" )
      R_Coil( "V3332_Xa_BonChua1" )
   END_RUNG
   // the same network as SCL:
   IF "PLC1_Manual_Mode_Active" AND NOT "V3332_Xa_BonChua1_Man" THEN "V3332_Xa_BonChua1" := FALSE; END_IF;
END_REGION

REGION Network 76: Manual V3333_DieuHuong_BonChua1 - Set
   RUNG wire#powerrail
      Contact( "PLC1_Manual_Mode_Active" )
      Contact( "V3333_DieuHuong_BonChua1_Man" )
      S_Coil( "V3333_DieuHuong_BonChua1" )
   END_RUNG
   // the same network as SCL:
   IF "PLC1_Manual_Mode_Active" AND "V3333_DieuHuong_BonChua1_Man" THEN
       "V3333_DieuHuong_BonChua1" := TRUE;
   END_IF;
END_REGION

REGION Network 77: Manual V3333_DieuHuong_BonChua1 - Reset
   RUNG wire#powerrail
      Contact( "PLC1_Manual_Mode_Active" )
      I_Contact( "V3333_DieuHuong_BonChua1_Man" )
      R_Coil( "V3333_DieuHuong_BonChua1" )
   END_RUNG
   // the same network as SCL:
   IF "PLC1_Manual_Mode_Active" AND NOT "V3333_DieuHuong_BonChua1_Man" THEN
       "V3333_DieuHuong_BonChua1" := FALSE;
   END_IF;
END_REGION

REGION Network 78: Manual V3334_DieuHuong_BonChua1 - Set
   RUNG wire#powerrail
      Contact( "PLC1_Manual_Mode_Active" )
      Contact( "V3334_DieuHuong_BonChua1_Man" )
      S_Coil( "V3334_DieuHuong_BonChua1" )
   END_RUNG
   // the same network as SCL:
   IF "PLC1_Manual_Mode_Active" AND "V3334_DieuHuong_BonChua1_Man" THEN
       "V3334_DieuHuong_BonChua1" := TRUE;
   END_IF;
END_REGION

REGION Network 79: Manual V3334_DieuHuong_BonChua1 - Reset
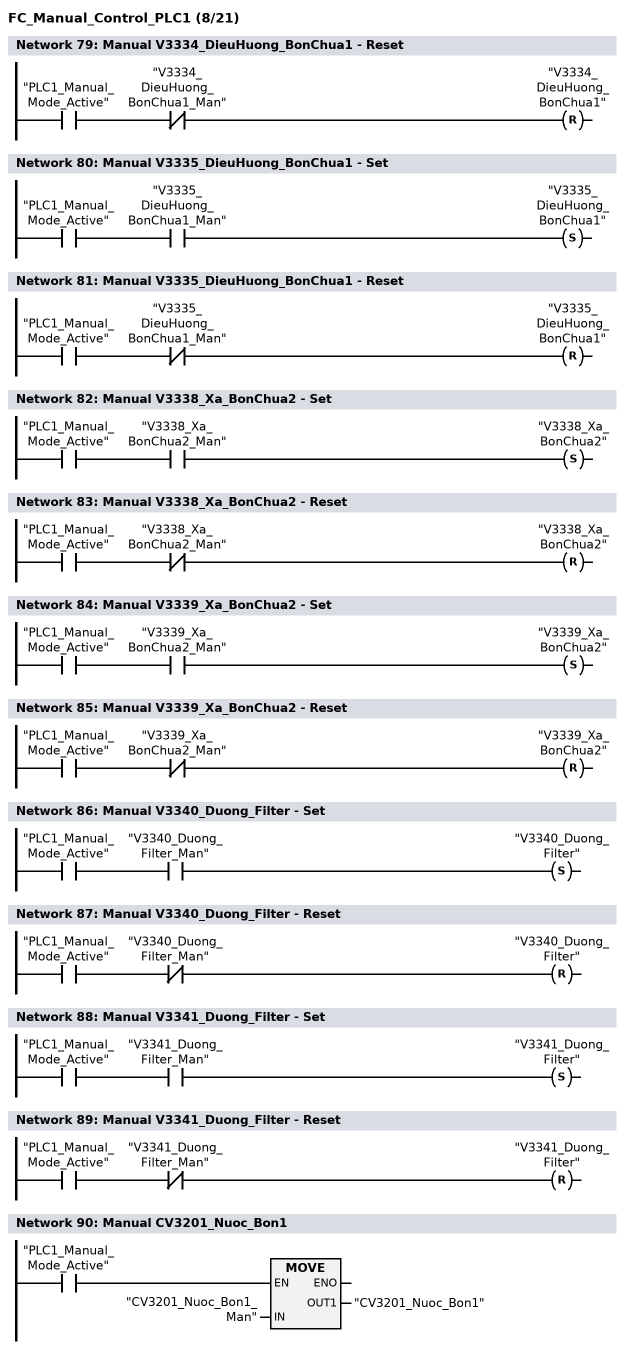
   RUNG wire#powerrail
      Contact( "PLC1_Manual_Mode_Active" )
      I_Contact( "V3334_DieuHuong_BonChua1_Man" )
      R_Coil( "V3334_DieuHuong_BonChua1" )
   END_RUNG
   // the same network as SCL:
   IF "PLC1_Manual_Mode_Active" AND NOT "V3334_DieuHuong_BonChua1_Man" THEN
       "V3334_DieuHuong_BonChua1" := FALSE;
   END_IF;
END_REGION

REGION Network 80: Manual V3335_DieuHuong_BonChua1 - Set
   RUNG wire#powerrail
      Contact( "PLC1_Manual_Mode_Active" )
      Contact( "V3335_DieuHuong_BonChua1_Man" )
      S_Coil( "V3335_DieuHuong_BonChua1" )
   END_RUNG
   // the same network as SCL:
   IF "PLC1_Manual_Mode_Active" AND "V3335_DieuHuong_BonChua1_Man" THEN
       "V3335_DieuHuong_BonChua1" := TRUE;
   END_IF;
END_REGION

REGION Network 81: Manual V3335_DieuHuong_BonChua1 - Reset
   RUNG wire#powerrail
      Contact( "PLC1_Manual_Mode_Active" )
      I_Contact( "V3335_DieuHuong_BonChua1_Man" )
      R_Coil( "V3335_DieuHuong_BonChua1" )
   END_RUNG
   // the same network as SCL:
   IF "PLC1_Manual_Mode_Active" AND NOT "V3335_DieuHuong_BonChua1_Man" THEN
       "V3335_DieuHuong_BonChua1" := FALSE;
   END_IF;
END_REGION

REGION Network 82: Manual V3338_Xa_BonChua2 - Set
   RUNG wire#powerrail
      Contact( "PLC1_Manual_Mode_Active" )
      Contact( "V3338_Xa_BonChua2_Man" )
      S_Coil( "V3338_Xa_BonChua2" )
   END_RUNG
   // the same network as SCL:
   IF "PLC1_Manual_Mode_Active" AND "V3338_Xa_BonChua2_Man" THEN "V3338_Xa_BonChua2" := TRUE; END_IF;
END_REGION

REGION Network 83: Manual V3338_Xa_BonChua2 - Reset
   RUNG wire#powerrail
      Contact( "PLC1_Manual_Mode_Active" )
      I_Contact( "V3338_Xa_BonChua2_Man" )
      R_Coil( "V3338_Xa_BonChua2" )
   END_RUNG
   // the same network as SCL:
   IF "PLC1_Manual_Mode_Active" AND NOT "V3338_Xa_BonChua2_Man" THEN "V3338_Xa_BonChua2" := FALSE; END_IF;
END_REGION

REGION Network 84: Manual V3339_Xa_BonChua2 - Set
   RUNG wire#powerrail
      Contact( "PLC1_Manual_Mode_Active" )
      Contact( "V3339_Xa_BonChua2_Man" )
      S_Coil( "V3339_Xa_BonChua2" )
   END_RUNG
   // the same network as SCL:
   IF "PLC1_Manual_Mode_Active" AND "V3339_Xa_BonChua2_Man" THEN "V3339_Xa_BonChua2" := TRUE; END_IF;
END_REGION

REGION Network 85: Manual V3339_Xa_BonChua2 - Reset
   RUNG wire#powerrail
      Contact( "PLC1_Manual_Mode_Active" )
      I_Contact( "V3339_Xa_BonChua2_Man" )
      R_Coil( "V3339_Xa_BonChua2" )
   END_RUNG
   // the same network as SCL:
   IF "PLC1_Manual_Mode_Active" AND NOT "V3339_Xa_BonChua2_Man" THEN "V3339_Xa_BonChua2" := FALSE; END_IF;
END_REGION

REGION Network 86: Manual V3340_Duong_Filter - Set
   RUNG wire#powerrail
      Contact( "PLC1_Manual_Mode_Active" )
      Contact( "V3340_Duong_Filter_Man" )
      S_Coil( "V3340_Duong_Filter" )
   END_RUNG
   // the same network as SCL:
   IF "PLC1_Manual_Mode_Active" AND "V3340_Duong_Filter_Man" THEN "V3340_Duong_Filter" := TRUE; END_IF;
END_REGION

REGION Network 87: Manual V3340_Duong_Filter - Reset
   RUNG wire#powerrail
      Contact( "PLC1_Manual_Mode_Active" )
      I_Contact( "V3340_Duong_Filter_Man" )
      R_Coil( "V3340_Duong_Filter" )
   END_RUNG
   // the same network as SCL:
   IF "PLC1_Manual_Mode_Active" AND NOT "V3340_Duong_Filter_Man" THEN "V3340_Duong_Filter" := FALSE; END_IF;
END_REGION

REGION Network 88: Manual V3341_Duong_Filter - Set
   RUNG wire#powerrail
      Contact( "PLC1_Manual_Mode_Active" )
      Contact( "V3341_Duong_Filter_Man" )
      S_Coil( "V3341_Duong_Filter" )
   END_RUNG
   // the same network as SCL:
   IF "PLC1_Manual_Mode_Active" AND "V3341_Duong_Filter_Man" THEN "V3341_Duong_Filter" := TRUE; END_IF;
END_REGION

REGION Network 89: Manual V3341_Duong_Filter - Reset
   RUNG wire#powerrail
      Contact( "PLC1_Manual_Mode_Active" )
      I_Contact( "V3341_Duong_Filter_Man" )
      R_Coil( "V3341_Duong_Filter" )
   END_RUNG
   // the same network as SCL:
   IF "PLC1_Manual_Mode_Active" AND NOT "V3341_Duong_Filter_Man" THEN "V3341_Duong_Filter" := FALSE; END_IF;
END_REGION

REGION Network 90: Manual CV3201_Nuoc_Bon1
   RUNG wire#powerrail
      Contact( "PLC1_Manual_Mode_Active" )
      { S7_GenerateENO := "TRUE" } Move(in := "CV3201_Nuoc_Bon1_Man", out1 => "CV3201_Nuoc_Bon1")
   END_RUNG
   // the same network as SCL:
   IF "PLC1_Manual_Mode_Active" THEN "CV3201_Nuoc_Bon1" := "CV3201_Nuoc_Bon1_Man"; END_IF;
END_REGION

REGION Network 91: Manual AGTR3260_Toc_Do_AO
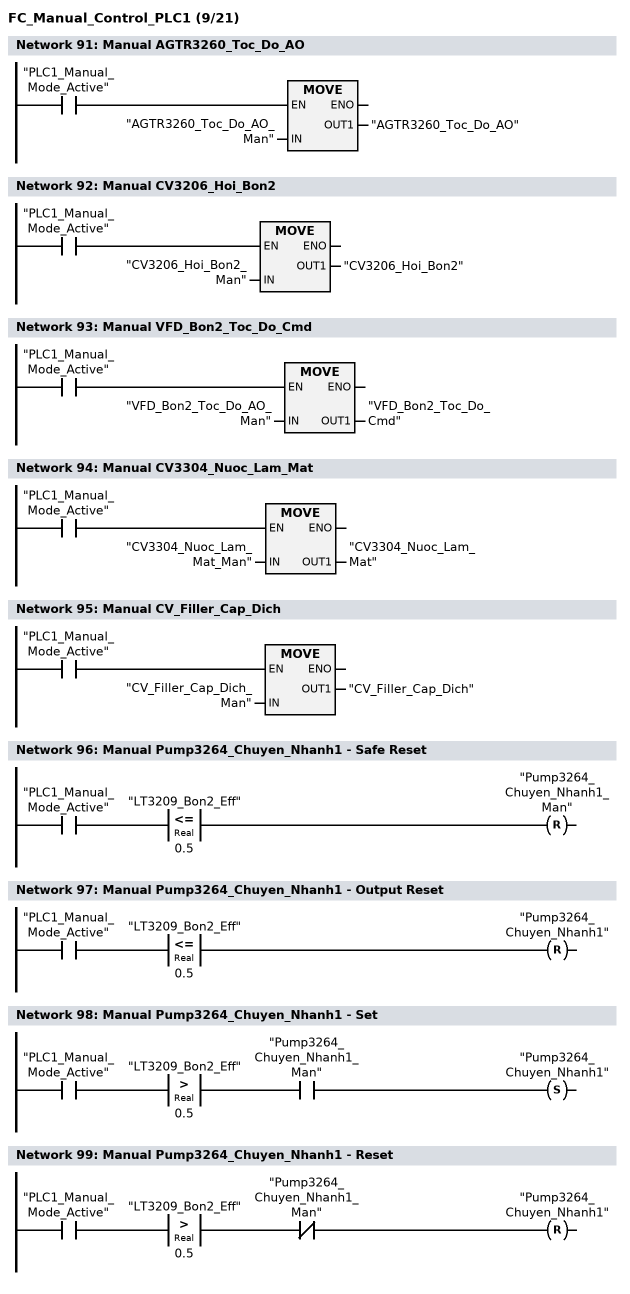
   RUNG wire#powerrail
      Contact( "PLC1_Manual_Mode_Active" )
      { S7_GenerateENO := "TRUE" } Move(in := "AGTR3260_Toc_Do_AO_Man", out1 => "AGTR3260_Toc_Do_AO")
   END_RUNG
   // the same network as SCL:
   IF "PLC1_Manual_Mode_Active" THEN "AGTR3260_Toc_Do_AO" := "AGTR3260_Toc_Do_AO_Man"; END_IF;
END_REGION

REGION Network 92: Manual CV3206_Hoi_Bon2
   RUNG wire#powerrail
      Contact( "PLC1_Manual_Mode_Active" )
      { S7_GenerateENO := "TRUE" } Move(in := "CV3206_Hoi_Bon2_Man", out1 => "CV3206_Hoi_Bon2")
   END_RUNG
   // the same network as SCL:
   IF "PLC1_Manual_Mode_Active" THEN "CV3206_Hoi_Bon2" := "CV3206_Hoi_Bon2_Man"; END_IF;
END_REGION

REGION Network 93: Manual VFD_Bon2_Toc_Do_Cmd
   RUNG wire#powerrail
      Contact( "PLC1_Manual_Mode_Active" )
      { S7_GenerateENO := "TRUE" } Move(in := "VFD_Bon2_Toc_Do_AO_Man", out1 => "VFD_Bon2_Toc_Do_Cmd")
   END_RUNG
   // the same network as SCL:
   IF "PLC1_Manual_Mode_Active" THEN "VFD_Bon2_Toc_Do_Cmd" := "VFD_Bon2_Toc_Do_AO_Man"; END_IF;
END_REGION

REGION Network 94: Manual CV3304_Nuoc_Lam_Mat
   RUNG wire#powerrail
      Contact( "PLC1_Manual_Mode_Active" )
      { S7_GenerateENO := "TRUE" } Move(in := "CV3304_Nuoc_Lam_Mat_Man", out1 => "CV3304_Nuoc_Lam_Mat")
   END_RUNG
   // the same network as SCL:
   IF "PLC1_Manual_Mode_Active" THEN "CV3304_Nuoc_Lam_Mat" := "CV3304_Nuoc_Lam_Mat_Man"; END_IF;
END_REGION

REGION Network 95: Manual CV_Filler_Cap_Dich
   RUNG wire#powerrail
      Contact( "PLC1_Manual_Mode_Active" )
      { S7_GenerateENO := "TRUE" } Move(in := "CV_Filler_Cap_Dich_Man", out1 => "CV_Filler_Cap_Dich")
   END_RUNG
   // the same network as SCL:
   IF "PLC1_Manual_Mode_Active" THEN "CV_Filler_Cap_Dich" := "CV_Filler_Cap_Dich_Man"; END_IF;
END_REGION

REGION Network 96: Manual Pump3264_Chuyen_Nhanh1 - Safe Reset
   RUNG wire#powerrail
      Contact( "PLC1_Manual_Mode_Active" )
      { S7_Templates := "SrcType := Real" } LE_Contact(in1 := "LT3209_Bon2_Eff", in2 := 0.5)
      R_Coil( "Pump3264_Chuyen_Nhanh1_Man" )
   END_RUNG
   // the same network as SCL:
   IF "PLC1_Manual_Mode_Active" AND ("LT3209_Bon2_Eff" <= 0.5) THEN
       "Pump3264_Chuyen_Nhanh1_Man" := FALSE;
   END_IF;
END_REGION

REGION Network 97: Manual Pump3264_Chuyen_Nhanh1 - Output Reset
   RUNG wire#powerrail
      Contact( "PLC1_Manual_Mode_Active" )
      { S7_Templates := "SrcType := Real" } LE_Contact(in1 := "LT3209_Bon2_Eff", in2 := 0.5)
      R_Coil( "Pump3264_Chuyen_Nhanh1" )
   END_RUNG
   // the same network as SCL:
   IF "PLC1_Manual_Mode_Active" AND ("LT3209_Bon2_Eff" <= 0.5) THEN
       "Pump3264_Chuyen_Nhanh1" := FALSE;
   END_IF;
END_REGION

REGION Network 98: Manual Pump3264_Chuyen_Nhanh1 - Set
   RUNG wire#powerrail
      Contact( "PLC1_Manual_Mode_Active" )
      { S7_Templates := "SrcType := Real" } GT_Contact(in1 := "LT3209_Bon2_Eff", in2 := 0.5)
      Contact( "Pump3264_Chuyen_Nhanh1_Man" )
      S_Coil( "Pump3264_Chuyen_Nhanh1" )
   END_RUNG
   // the same network as SCL:
   IF "PLC1_Manual_Mode_Active" AND ("LT3209_Bon2_Eff" > 0.5) AND "Pump3264_Chuyen_Nhanh1_Man" THEN
       "Pump3264_Chuyen_Nhanh1" := TRUE;
   END_IF;
END_REGION

REGION Network 99: Manual Pump3264_Chuyen_Nhanh1 - Reset
   RUNG wire#powerrail
      Contact( "PLC1_Manual_Mode_Active" )
      { S7_Templates := "SrcType := Real" } GT_Contact(in1 := "LT3209_Bon2_Eff", in2 := 0.5)
      I_Contact( "Pump3264_Chuyen_Nhanh1_Man" )
      R_Coil( "Pump3264_Chuyen_Nhanh1" )
   END_RUNG
   // the same network as SCL:
   IF "PLC1_Manual_Mode_Active" AND ("LT3209_Bon2_Eff" > 0.5) AND NOT "Pump3264_Chuyen_Nhanh1_Man" THEN
       "Pump3264_Chuyen_Nhanh1" := FALSE;
   END_IF;
END_REGION

REGION Network 100: Manual Pump3361_LuanChuyen_BonChua1 - Safe Reset
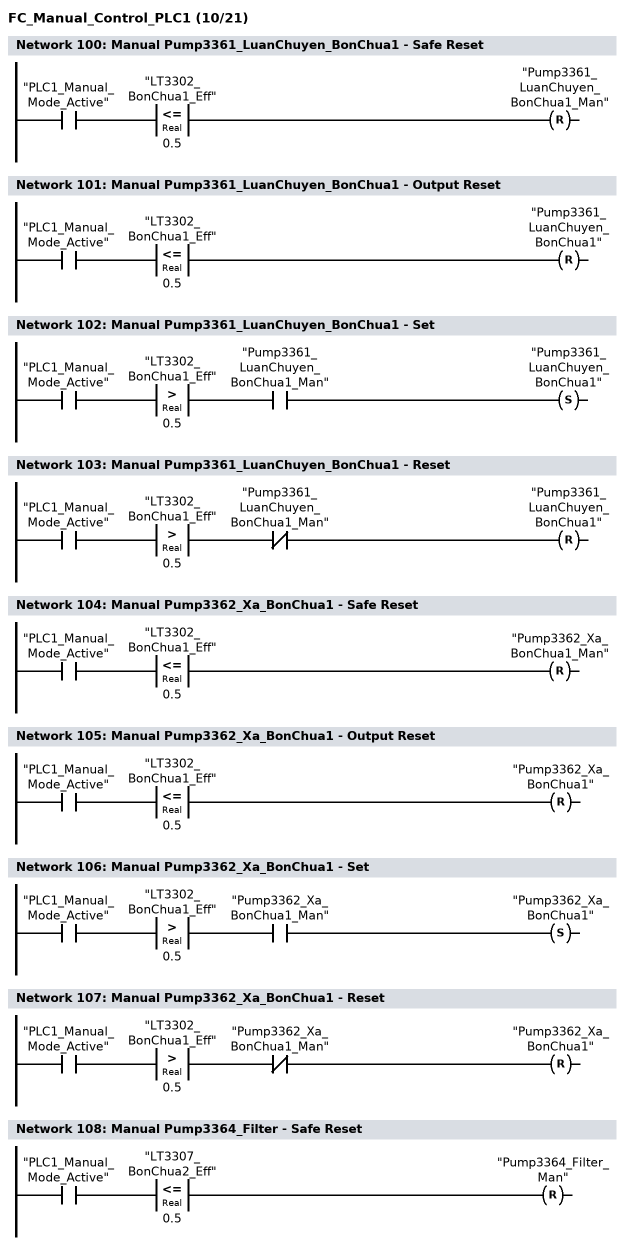
   RUNG wire#powerrail
      Contact( "PLC1_Manual_Mode_Active" )
      { S7_Templates := "SrcType := Real" } LE_Contact(in1 := "LT3302_BonChua1_Eff", in2 := 0.5)
      R_Coil( "Pump3361_LuanChuyen_BonChua1_Man" )
   END_RUNG
   // the same network as SCL:
   IF "PLC1_Manual_Mode_Active" AND ("LT3302_BonChua1_Eff" <= 0.5) THEN
       "Pump3361_LuanChuyen_BonChua1_Man" := FALSE;
   END_IF;
END_REGION

REGION Network 101: Manual Pump3361_LuanChuyen_BonChua1 - Output Reset
   RUNG wire#powerrail
      Contact( "PLC1_Manual_Mode_Active" )
      { S7_Templates := "SrcType := Real" } LE_Contact(in1 := "LT3302_BonChua1_Eff", in2 := 0.5)
      R_Coil( "Pump3361_LuanChuyen_BonChua1" )
   END_RUNG
   // the same network as SCL:
   IF "PLC1_Manual_Mode_Active" AND ("LT3302_BonChua1_Eff" <= 0.5) THEN
       "Pump3361_LuanChuyen_BonChua1" := FALSE;
   END_IF;
END_REGION

REGION Network 102: Manual Pump3361_LuanChuyen_BonChua1 - Set
   RUNG wire#powerrail
      Contact( "PLC1_Manual_Mode_Active" )
      { S7_Templates := "SrcType := Real" } GT_Contact(in1 := "LT3302_BonChua1_Eff", in2 := 0.5)
      Contact( "Pump3361_LuanChuyen_BonChua1_Man" )
      S_Coil( "Pump3361_LuanChuyen_BonChua1" )
   END_RUNG
   // the same network as SCL:
   IF "PLC1_Manual_Mode_Active" AND ("LT3302_BonChua1_Eff" > 0.5) AND "Pump3361_LuanChuyen_BonChua1_Man" THEN
       "Pump3361_LuanChuyen_BonChua1" := TRUE;
   END_IF;
END_REGION

REGION Network 103: Manual Pump3361_LuanChuyen_BonChua1 - Reset
   RUNG wire#powerrail
      Contact( "PLC1_Manual_Mode_Active" )
      { S7_Templates := "SrcType := Real" } GT_Contact(in1 := "LT3302_BonChua1_Eff", in2 := 0.5)
      I_Contact( "Pump3361_LuanChuyen_BonChua1_Man" )
      R_Coil( "Pump3361_LuanChuyen_BonChua1" )
   END_RUNG
   // the same network as SCL:
   IF "PLC1_Manual_Mode_Active" AND ("LT3302_BonChua1_Eff" > 0.5) AND NOT "Pump3361_LuanChuyen_BonChua1_Man" THEN
       "Pump3361_LuanChuyen_BonChua1" := FALSE;
   END_IF;
END_REGION

REGION Network 104: Manual Pump3362_Xa_BonChua1 - Safe Reset
   RUNG wire#powerrail
      Contact( "PLC1_Manual_Mode_Active" )
      { S7_Templates := "SrcType := Real" } LE_Contact(in1 := "LT3302_BonChua1_Eff", in2 := 0.5)
      R_Coil( "Pump3362_Xa_BonChua1_Man" )
   END_RUNG
   // the same network as SCL:
   IF "PLC1_Manual_Mode_Active" AND ("LT3302_BonChua1_Eff" <= 0.5) THEN
       "Pump3362_Xa_BonChua1_Man" := FALSE;
   END_IF;
END_REGION

REGION Network 105: Manual Pump3362_Xa_BonChua1 - Output Reset
   RUNG wire#powerrail
      Contact( "PLC1_Manual_Mode_Active" )
      { S7_Templates := "SrcType := Real" } LE_Contact(in1 := "LT3302_BonChua1_Eff", in2 := 0.5)
      R_Coil( "Pump3362_Xa_BonChua1" )
   END_RUNG
   // the same network as SCL:
   IF "PLC1_Manual_Mode_Active" AND ("LT3302_BonChua1_Eff" <= 0.5) THEN
       "Pump3362_Xa_BonChua1" := FALSE;
   END_IF;
END_REGION

REGION Network 106: Manual Pump3362_Xa_BonChua1 - Set
   RUNG wire#powerrail
      Contact( "PLC1_Manual_Mode_Active" )
      { S7_Templates := "SrcType := Real" } GT_Contact(in1 := "LT3302_BonChua1_Eff", in2 := 0.5)
      Contact( "Pump3362_Xa_BonChua1_Man" )
      S_Coil( "Pump3362_Xa_BonChua1" )
   END_RUNG
   // the same network as SCL:
   IF "PLC1_Manual_Mode_Active" AND ("LT3302_BonChua1_Eff" > 0.5) AND "Pump3362_Xa_BonChua1_Man" THEN
       "Pump3362_Xa_BonChua1" := TRUE;
   END_IF;
END_REGION

REGION Network 107: Manual Pump3362_Xa_BonChua1 - Reset
   RUNG wire#powerrail
      Contact( "PLC1_Manual_Mode_Active" )
      { S7_Templates := "SrcType := Real" } GT_Contact(in1 := "LT3302_BonChua1_Eff", in2 := 0.5)
      I_Contact( "Pump3362_Xa_BonChua1_Man" )
      R_Coil( "Pump3362_Xa_BonChua1" )
   END_RUNG
   // the same network as SCL:
   IF "PLC1_Manual_Mode_Active" AND ("LT3302_BonChua1_Eff" > 0.5) AND NOT "Pump3362_Xa_BonChua1_Man" THEN
       "Pump3362_Xa_BonChua1" := FALSE;
   END_IF;
END_REGION

REGION Network 108: Manual Pump3364_Filter - Safe Reset
   RUNG wire#powerrail
      Contact( "PLC1_Manual_Mode_Active" )
      { S7_Templates := "SrcType := Real" } LE_Contact(in1 := "LT3307_BonChua2_Eff", in2 := 0.5)
      R_Coil( "Pump3364_Filter_Man" )
   END_RUNG
   // the same network as SCL:
   IF "PLC1_Manual_Mode_Active" AND ("LT3307_BonChua2_Eff" <= 0.5) THEN
       "Pump3364_Filter_Man" := FALSE;
   END_IF;
END_REGION

REGION Network 109: Manual Pump3364_Filter - Output Reset
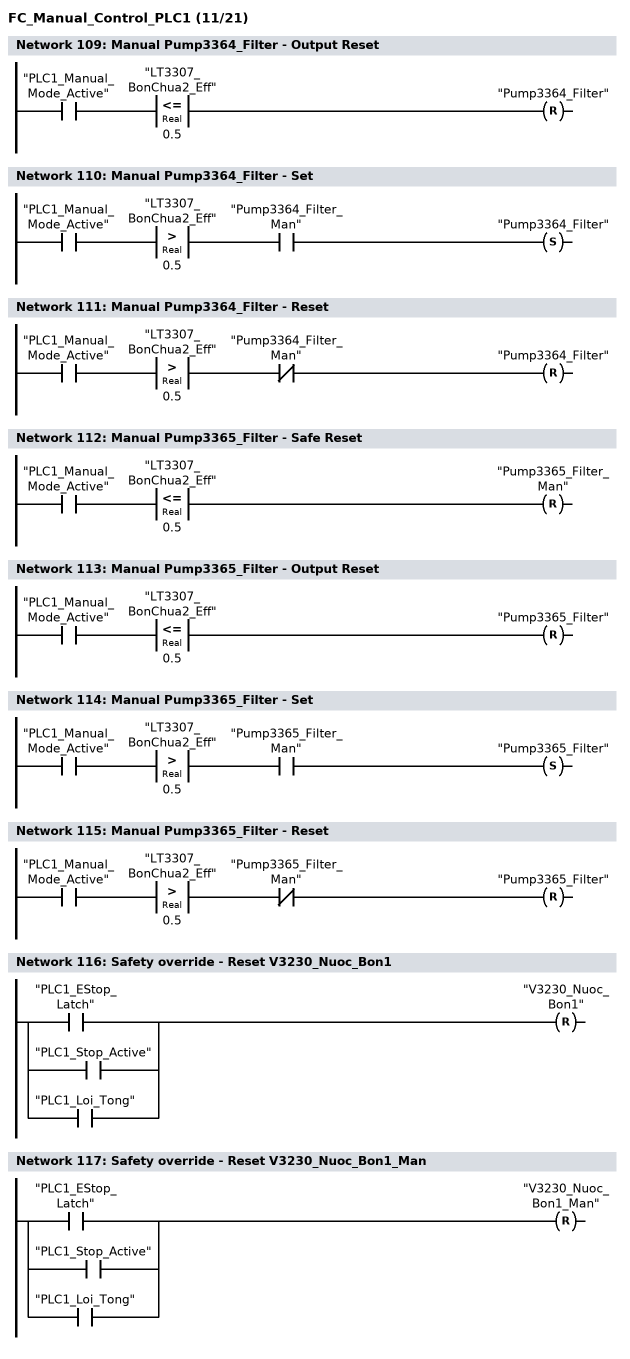
   RUNG wire#powerrail
      Contact( "PLC1_Manual_Mode_Active" )
      { S7_Templates := "SrcType := Real" } LE_Contact(in1 := "LT3307_BonChua2_Eff", in2 := 0.5)
      R_Coil( "Pump3364_Filter" )
   END_RUNG
   // the same network as SCL:
   IF "PLC1_Manual_Mode_Active" AND ("LT3307_BonChua2_Eff" <= 0.5) THEN "Pump3364_Filter" := FALSE; END_IF;
END_REGION

REGION Network 110: Manual Pump3364_Filter - Set
   RUNG wire#powerrail
      Contact( "PLC1_Manual_Mode_Active" )
      { S7_Templates := "SrcType := Real" } GT_Contact(in1 := "LT3307_BonChua2_Eff", in2 := 0.5)
      Contact( "Pump3364_Filter_Man" )
      S_Coil( "Pump3364_Filter" )
   END_RUNG
   // the same network as SCL:
   IF "PLC1_Manual_Mode_Active" AND ("LT3307_BonChua2_Eff" > 0.5) AND "Pump3364_Filter_Man" THEN
       "Pump3364_Filter" := TRUE;
   END_IF;
END_REGION

REGION Network 111: Manual Pump3364_Filter - Reset
   RUNG wire#powerrail
      Contact( "PLC1_Manual_Mode_Active" )
      { S7_Templates := "SrcType := Real" } GT_Contact(in1 := "LT3307_BonChua2_Eff", in2 := 0.5)
      I_Contact( "Pump3364_Filter_Man" )
      R_Coil( "Pump3364_Filter" )
   END_RUNG
   // the same network as SCL:
   IF "PLC1_Manual_Mode_Active" AND ("LT3307_BonChua2_Eff" > 0.5) AND NOT "Pump3364_Filter_Man" THEN
       "Pump3364_Filter" := FALSE;
   END_IF;
END_REGION

REGION Network 112: Manual Pump3365_Filter - Safe Reset
   RUNG wire#powerrail
      Contact( "PLC1_Manual_Mode_Active" )
      { S7_Templates := "SrcType := Real" } LE_Contact(in1 := "LT3307_BonChua2_Eff", in2 := 0.5)
      R_Coil( "Pump3365_Filter_Man" )
   END_RUNG
   // the same network as SCL:
   IF "PLC1_Manual_Mode_Active" AND ("LT3307_BonChua2_Eff" <= 0.5) THEN
       "Pump3365_Filter_Man" := FALSE;
   END_IF;
END_REGION

REGION Network 113: Manual Pump3365_Filter - Output Reset
   RUNG wire#powerrail
      Contact( "PLC1_Manual_Mode_Active" )
      { S7_Templates := "SrcType := Real" } LE_Contact(in1 := "LT3307_BonChua2_Eff", in2 := 0.5)
      R_Coil( "Pump3365_Filter" )
   END_RUNG
   // the same network as SCL:
   IF "PLC1_Manual_Mode_Active" AND ("LT3307_BonChua2_Eff" <= 0.5) THEN "Pump3365_Filter" := FALSE; END_IF;
END_REGION

REGION Network 114: Manual Pump3365_Filter - Set
   RUNG wire#powerrail
      Contact( "PLC1_Manual_Mode_Active" )
      { S7_Templates := "SrcType := Real" } GT_Contact(in1 := "LT3307_BonChua2_Eff", in2 := 0.5)
      Contact( "Pump3365_Filter_Man" )
      S_Coil( "Pump3365_Filter" )
   END_RUNG
   // the same network as SCL:
   IF "PLC1_Manual_Mode_Active" AND ("LT3307_BonChua2_Eff" > 0.5) AND "Pump3365_Filter_Man" THEN
       "Pump3365_Filter" := TRUE;
   END_IF;
END_REGION

REGION Network 115: Manual Pump3365_Filter - Reset
   RUNG wire#powerrail
      Contact( "PLC1_Manual_Mode_Active" )
      { S7_Templates := "SrcType := Real" } GT_Contact(in1 := "LT3307_BonChua2_Eff", in2 := 0.5)
      I_Contact( "Pump3365_Filter_Man" )
      R_Coil( "Pump3365_Filter" )
   END_RUNG
   // the same network as SCL:
   IF "PLC1_Manual_Mode_Active" AND ("LT3307_BonChua2_Eff" > 0.5) AND NOT "Pump3365_Filter_Man" THEN
       "Pump3365_Filter" := FALSE;
   END_IF;
END_REGION

REGION Network 116: Safety override - Reset V3230_Nuoc_Bon1
   RUNG wire#powerrail
      Contact( "PLC1_EStop_Latch" )
      wire#w1
      R_Coil( "V3230_Nuoc_Bon1" )
   END_RUNG
   RUNG wire#powerrail
      Contact( "PLC1_Stop_Active" )
   END_RUNG wire#w1
   RUNG wire#powerrail
      Contact( "PLC1_Loi_Tong" )
   END_RUNG wire#w1
   // the same network as SCL:
   IF "PLC1_EStop_Latch" OR "PLC1_Stop_Active" OR "PLC1_Loi_Tong" THEN "V3230_Nuoc_Bon1" := FALSE; END_IF;
END_REGION

REGION Network 117: Safety override - Reset V3230_Nuoc_Bon1_Man
   RUNG wire#powerrail
      Contact( "PLC1_EStop_Latch" )
      wire#w1
      R_Coil( "V3230_Nuoc_Bon1_Man" )
   END_RUNG
   RUNG wire#powerrail
      Contact( "PLC1_Stop_Active" )
   END_RUNG wire#w1
   RUNG wire#powerrail
      Contact( "PLC1_Loi_Tong" )
   END_RUNG wire#w1
   // the same network as SCL:
   IF "PLC1_EStop_Latch" OR "PLC1_Stop_Active" OR "PLC1_Loi_Tong" THEN
       "V3230_Nuoc_Bon1_Man" := FALSE;
   END_IF;
END_REGION

REGION Network 118: Safety override - Reset AGTR3260_Khuay_Bon1
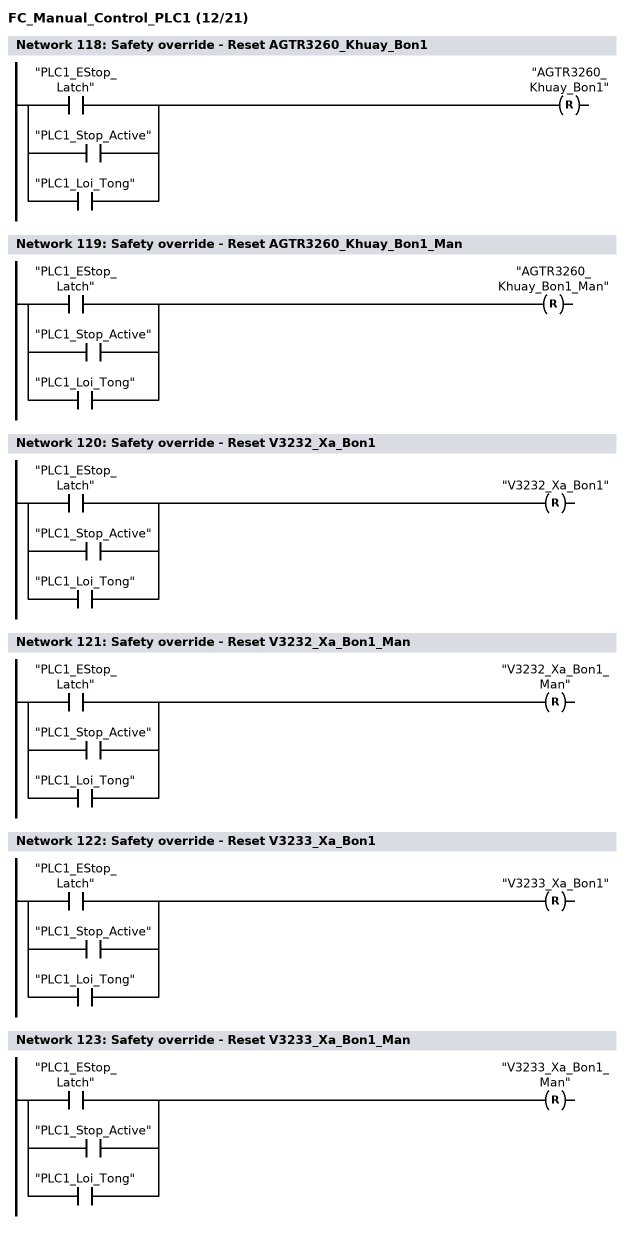
   RUNG wire#powerrail
      Contact( "PLC1_EStop_Latch" )
      wire#w1
      R_Coil( "AGTR3260_Khuay_Bon1" )
   END_RUNG
   RUNG wire#powerrail
      Contact( "PLC1_Stop_Active" )
   END_RUNG wire#w1
   RUNG wire#powerrail
      Contact( "PLC1_Loi_Tong" )
   END_RUNG wire#w1
   // the same network as SCL:
   IF "PLC1_EStop_Latch" OR "PLC1_Stop_Active" OR "PLC1_Loi_Tong" THEN
       "AGTR3260_Khuay_Bon1" := FALSE;
   END_IF;
END_REGION

REGION Network 119: Safety override - Reset AGTR3260_Khuay_Bon1_Man
   RUNG wire#powerrail
      Contact( "PLC1_EStop_Latch" )
      wire#w1
      R_Coil( "AGTR3260_Khuay_Bon1_Man" )
   END_RUNG
   RUNG wire#powerrail
      Contact( "PLC1_Stop_Active" )
   END_RUNG wire#w1
   RUNG wire#powerrail
      Contact( "PLC1_Loi_Tong" )
   END_RUNG wire#w1
   // the same network as SCL:
   IF "PLC1_EStop_Latch" OR "PLC1_Stop_Active" OR "PLC1_Loi_Tong" THEN
       "AGTR3260_Khuay_Bon1_Man" := FALSE;
   END_IF;
END_REGION

REGION Network 120: Safety override - Reset V3232_Xa_Bon1
   RUNG wire#powerrail
      Contact( "PLC1_EStop_Latch" )
      wire#w1
      R_Coil( "V3232_Xa_Bon1" )
   END_RUNG
   RUNG wire#powerrail
      Contact( "PLC1_Stop_Active" )
   END_RUNG wire#w1
   RUNG wire#powerrail
      Contact( "PLC1_Loi_Tong" )
   END_RUNG wire#w1
   // the same network as SCL:
   IF "PLC1_EStop_Latch" OR "PLC1_Stop_Active" OR "PLC1_Loi_Tong" THEN "V3232_Xa_Bon1" := FALSE; END_IF;
END_REGION

REGION Network 121: Safety override - Reset V3232_Xa_Bon1_Man
   RUNG wire#powerrail
      Contact( "PLC1_EStop_Latch" )
      wire#w1
      R_Coil( "V3232_Xa_Bon1_Man" )
   END_RUNG
   RUNG wire#powerrail
      Contact( "PLC1_Stop_Active" )
   END_RUNG wire#w1
   RUNG wire#powerrail
      Contact( "PLC1_Loi_Tong" )
   END_RUNG wire#w1
   // the same network as SCL:
   IF "PLC1_EStop_Latch" OR "PLC1_Stop_Active" OR "PLC1_Loi_Tong" THEN "V3232_Xa_Bon1_Man" := FALSE; END_IF;
END_REGION

REGION Network 122: Safety override - Reset V3233_Xa_Bon1
   RUNG wire#powerrail
      Contact( "PLC1_EStop_Latch" )
      wire#w1
      R_Coil( "V3233_Xa_Bon1" )
   END_RUNG
   RUNG wire#powerrail
      Contact( "PLC1_Stop_Active" )
   END_RUNG wire#w1
   RUNG wire#powerrail
      Contact( "PLC1_Loi_Tong" )
   END_RUNG wire#w1
   // the same network as SCL:
   IF "PLC1_EStop_Latch" OR "PLC1_Stop_Active" OR "PLC1_Loi_Tong" THEN "V3233_Xa_Bon1" := FALSE; END_IF;
END_REGION

REGION Network 123: Safety override - Reset V3233_Xa_Bon1_Man
   RUNG wire#powerrail
      Contact( "PLC1_EStop_Latch" )
      wire#w1
      R_Coil( "V3233_Xa_Bon1_Man" )
   END_RUNG
   RUNG wire#powerrail
      Contact( "PLC1_Stop_Active" )
   END_RUNG wire#w1
   RUNG wire#powerrail
      Contact( "PLC1_Loi_Tong" )
   END_RUNG wire#w1
   // the same network as SCL:
   IF "PLC1_EStop_Latch" OR "PLC1_Stop_Active" OR "PLC1_Loi_Tong" THEN "V3233_Xa_Bon1_Man" := FALSE; END_IF;
END_REGION

REGION Network 124: Safety override - Reset V3234_Xa_Bon1
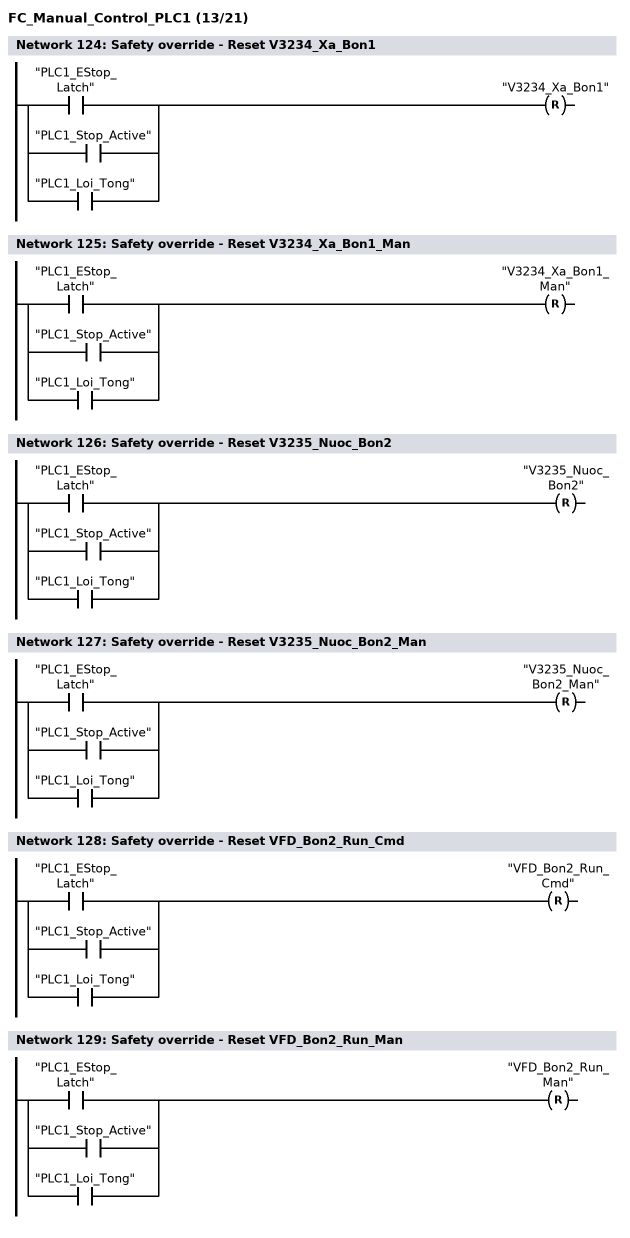
   RUNG wire#powerrail
      Contact( "PLC1_EStop_Latch" )
      wire#w1
      R_Coil( "V3234_Xa_Bon1" )
   END_RUNG
   RUNG wire#powerrail
      Contact( "PLC1_Stop_Active" )
   END_RUNG wire#w1
   RUNG wire#powerrail
      Contact( "PLC1_Loi_Tong" )
   END_RUNG wire#w1
   // the same network as SCL:
   IF "PLC1_EStop_Latch" OR "PLC1_Stop_Active" OR "PLC1_Loi_Tong" THEN "V3234_Xa_Bon1" := FALSE; END_IF;
END_REGION

REGION Network 125: Safety override - Reset V3234_Xa_Bon1_Man
   RUNG wire#powerrail
      Contact( "PLC1_EStop_Latch" )
      wire#w1
      R_Coil( "V3234_Xa_Bon1_Man" )
   END_RUNG
   RUNG wire#powerrail
      Contact( "PLC1_Stop_Active" )
   END_RUNG wire#w1
   RUNG wire#powerrail
      Contact( "PLC1_Loi_Tong" )
   END_RUNG wire#w1
   // the same network as SCL:
   IF "PLC1_EStop_Latch" OR "PLC1_Stop_Active" OR "PLC1_Loi_Tong" THEN "V3234_Xa_Bon1_Man" := FALSE; END_IF;
END_REGION

REGION Network 126: Safety override - Reset V3235_Nuoc_Bon2
   RUNG wire#powerrail
      Contact( "PLC1_EStop_Latch" )
      wire#w1
      R_Coil( "V3235_Nuoc_Bon2" )
   END_RUNG
   RUNG wire#powerrail
      Contact( "PLC1_Stop_Active" )
   END_RUNG wire#w1
   RUNG wire#powerrail
      Contact( "PLC1_Loi_Tong" )
   END_RUNG wire#w1
   // the same network as SCL:
   IF "PLC1_EStop_Latch" OR "PLC1_Stop_Active" OR "PLC1_Loi_Tong" THEN "V3235_Nuoc_Bon2" := FALSE; END_IF;
END_REGION

REGION Network 127: Safety override - Reset V3235_Nuoc_Bon2_Man
   RUNG wire#powerrail
      Contact( "PLC1_EStop_Latch" )
      wire#w1
      R_Coil( "V3235_Nuoc_Bon2_Man" )
   END_RUNG
   RUNG wire#powerrail
      Contact( "PLC1_Stop_Active" )
   END_RUNG wire#w1
   RUNG wire#powerrail
      Contact( "PLC1_Loi_Tong" )
   END_RUNG wire#w1
   // the same network as SCL:
   IF "PLC1_EStop_Latch" OR "PLC1_Stop_Active" OR "PLC1_Loi_Tong" THEN
       "V3235_Nuoc_Bon2_Man" := FALSE;
   END_IF;
END_REGION

REGION Network 128: Safety override - Reset VFD_Bon2_Run_Cmd
   RUNG wire#powerrail
      Contact( "PLC1_EStop_Latch" )
      wire#w1
      R_Coil( "VFD_Bon2_Run_Cmd" )
   END_RUNG
   RUNG wire#powerrail
      Contact( "PLC1_Stop_Active" )
   END_RUNG wire#w1
   RUNG wire#powerrail
      Contact( "PLC1_Loi_Tong" )
   END_RUNG wire#w1
   // the same network as SCL:
   IF "PLC1_EStop_Latch" OR "PLC1_Stop_Active" OR "PLC1_Loi_Tong" THEN "VFD_Bon2_Run_Cmd" := FALSE; END_IF;
END_REGION

REGION Network 129: Safety override - Reset VFD_Bon2_Run_Man
   RUNG wire#powerrail
      Contact( "PLC1_EStop_Latch" )
      wire#w1
      R_Coil( "VFD_Bon2_Run_Man" )
   END_RUNG
   RUNG wire#powerrail
      Contact( "PLC1_Stop_Active" )
   END_RUNG wire#w1
   RUNG wire#powerrail
      Contact( "PLC1_Loi_Tong" )
   END_RUNG wire#w1
   // the same network as SCL:
   IF "PLC1_EStop_Latch" OR "PLC1_Stop_Active" OR "PLC1_Loi_Tong" THEN "VFD_Bon2_Run_Man" := FALSE; END_IF;
END_REGION

REGION Network 130: Safety override - Reset VFD_Bon2_Dao_Chieu_Cmd
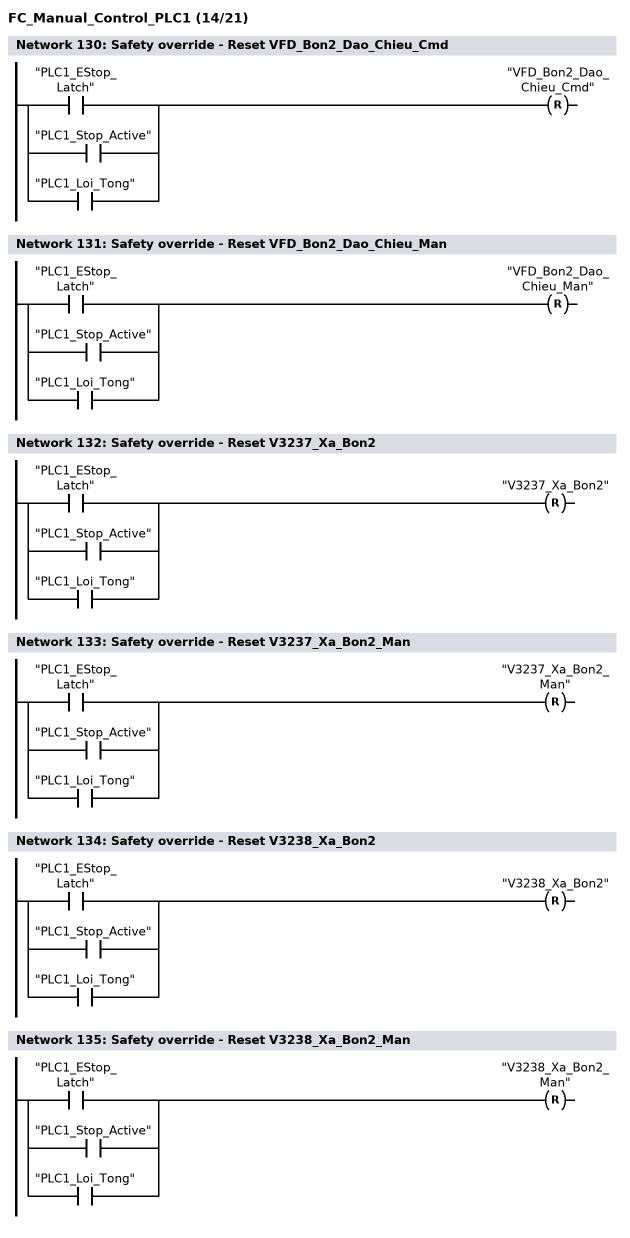
   RUNG wire#powerrail
      Contact( "PLC1_EStop_Latch" )
      wire#w1
      R_Coil( "VFD_Bon2_Dao_Chieu_Cmd" )
   END_RUNG
   RUNG wire#powerrail
      Contact( "PLC1_Stop_Active" )
   END_RUNG wire#w1
   RUNG wire#powerrail
      Contact( "PLC1_Loi_Tong" )
   END_RUNG wire#w1
   // the same network as SCL:
   IF "PLC1_EStop_Latch" OR "PLC1_Stop_Active" OR "PLC1_Loi_Tong" THEN
       "VFD_Bon2_Dao_Chieu_Cmd" := FALSE;
   END_IF;
END_REGION

REGION Network 131: Safety override - Reset VFD_Bon2_Dao_Chieu_Man
   RUNG wire#powerrail
      Contact( "PLC1_EStop_Latch" )
      wire#w1
      R_Coil( "VFD_Bon2_Dao_Chieu_Man" )
   END_RUNG
   RUNG wire#powerrail
      Contact( "PLC1_Stop_Active" )
   END_RUNG wire#w1
   RUNG wire#powerrail
      Contact( "PLC1_Loi_Tong" )
   END_RUNG wire#w1
   // the same network as SCL:
   IF "PLC1_EStop_Latch" OR "PLC1_Stop_Active" OR "PLC1_Loi_Tong" THEN
       "VFD_Bon2_Dao_Chieu_Man" := FALSE;
   END_IF;
END_REGION

REGION Network 132: Safety override - Reset V3237_Xa_Bon2
   RUNG wire#powerrail
      Contact( "PLC1_EStop_Latch" )
      wire#w1
      R_Coil( "V3237_Xa_Bon2" )
   END_RUNG
   RUNG wire#powerrail
      Contact( "PLC1_Stop_Active" )
   END_RUNG wire#w1
   RUNG wire#powerrail
      Contact( "PLC1_Loi_Tong" )
   END_RUNG wire#w1
   // the same network as SCL:
   IF "PLC1_EStop_Latch" OR "PLC1_Stop_Active" OR "PLC1_Loi_Tong" THEN "V3237_Xa_Bon2" := FALSE; END_IF;
END_REGION

REGION Network 133: Safety override - Reset V3237_Xa_Bon2_Man
   RUNG wire#powerrail
      Contact( "PLC1_EStop_Latch" )
      wire#w1
      R_Coil( "V3237_Xa_Bon2_Man" )
   END_RUNG
   RUNG wire#powerrail
      Contact( "PLC1_Stop_Active" )
   END_RUNG wire#w1
   RUNG wire#powerrail
      Contact( "PLC1_Loi_Tong" )
   END_RUNG wire#w1
   // the same network as SCL:
   IF "PLC1_EStop_Latch" OR "PLC1_Stop_Active" OR "PLC1_Loi_Tong" THEN "V3237_Xa_Bon2_Man" := FALSE; END_IF;
END_REGION

REGION Network 134: Safety override - Reset V3238_Xa_Bon2
   RUNG wire#powerrail
      Contact( "PLC1_EStop_Latch" )
      wire#w1
      R_Coil( "V3238_Xa_Bon2" )
   END_RUNG
   RUNG wire#powerrail
      Contact( "PLC1_Stop_Active" )
   END_RUNG wire#w1
   RUNG wire#powerrail
      Contact( "PLC1_Loi_Tong" )
   END_RUNG wire#w1
   // the same network as SCL:
   IF "PLC1_EStop_Latch" OR "PLC1_Stop_Active" OR "PLC1_Loi_Tong" THEN "V3238_Xa_Bon2" := FALSE; END_IF;
END_REGION

REGION Network 135: Safety override - Reset V3238_Xa_Bon2_Man
   RUNG wire#powerrail
      Contact( "PLC1_EStop_Latch" )
      wire#w1
      R_Coil( "V3238_Xa_Bon2_Man" )
   END_RUNG
   RUNG wire#powerrail
      Contact( "PLC1_Stop_Active" )
   END_RUNG wire#w1
   RUNG wire#powerrail
      Contact( "PLC1_Loi_Tong" )
   END_RUNG wire#w1
   // the same network as SCL:
   IF "PLC1_EStop_Latch" OR "PLC1_Stop_Active" OR "PLC1_Loi_Tong" THEN "V3238_Xa_Bon2_Man" := FALSE; END_IF;
END_REGION

REGION Network 136: Safety override - Reset V3239_Xa_Bon2
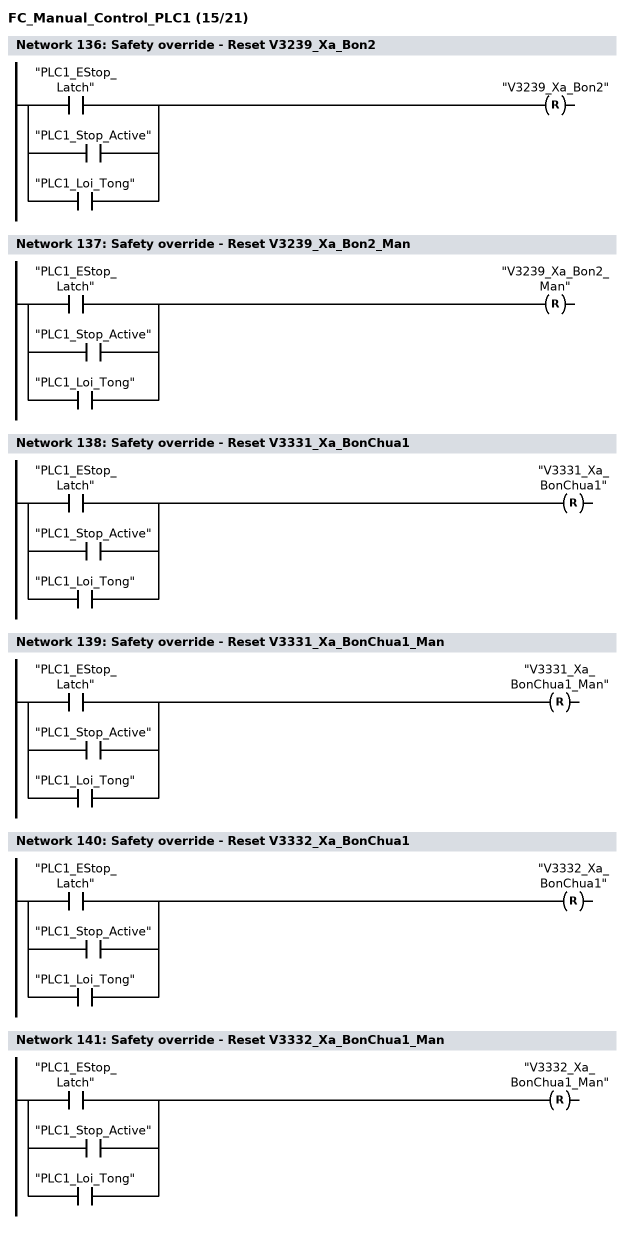
   RUNG wire#powerrail
      Contact( "PLC1_EStop_Latch" )
      wire#w1
      R_Coil( "V3239_Xa_Bon2" )
   END_RUNG
   RUNG wire#powerrail
      Contact( "PLC1_Stop_Active" )
   END_RUNG wire#w1
   RUNG wire#powerrail
      Contact( "PLC1_Loi_Tong" )
   END_RUNG wire#w1
   // the same network as SCL:
   IF "PLC1_EStop_Latch" OR "PLC1_Stop_Active" OR "PLC1_Loi_Tong" THEN "V3239_Xa_Bon2" := FALSE; END_IF;
END_REGION

REGION Network 137: Safety override - Reset V3239_Xa_Bon2_Man
   RUNG wire#powerrail
      Contact( "PLC1_EStop_Latch" )
      wire#w1
      R_Coil( "V3239_Xa_Bon2_Man" )
   END_RUNG
   RUNG wire#powerrail
      Contact( "PLC1_Stop_Active" )
   END_RUNG wire#w1
   RUNG wire#powerrail
      Contact( "PLC1_Loi_Tong" )
   END_RUNG wire#w1
   // the same network as SCL:
   IF "PLC1_EStop_Latch" OR "PLC1_Stop_Active" OR "PLC1_Loi_Tong" THEN "V3239_Xa_Bon2_Man" := FALSE; END_IF;
END_REGION

REGION Network 138: Safety override - Reset V3331_Xa_BonChua1
   RUNG wire#powerrail
      Contact( "PLC1_EStop_Latch" )
      wire#w1
      R_Coil( "V3331_Xa_BonChua1" )
   END_RUNG
   RUNG wire#powerrail
      Contact( "PLC1_Stop_Active" )
   END_RUNG wire#w1
   RUNG wire#powerrail
      Contact( "PLC1_Loi_Tong" )
   END_RUNG wire#w1
   // the same network as SCL:
   IF "PLC1_EStop_Latch" OR "PLC1_Stop_Active" OR "PLC1_Loi_Tong" THEN "V3331_Xa_BonChua1" := FALSE; END_IF;
END_REGION

REGION Network 139: Safety override - Reset V3331_Xa_BonChua1_Man
   RUNG wire#powerrail
      Contact( "PLC1_EStop_Latch" )
      wire#w1
      R_Coil( "V3331_Xa_BonChua1_Man" )
   END_RUNG
   RUNG wire#powerrail
      Contact( "PLC1_Stop_Active" )
   END_RUNG wire#w1
   RUNG wire#powerrail
      Contact( "PLC1_Loi_Tong" )
   END_RUNG wire#w1
   // the same network as SCL:
   IF "PLC1_EStop_Latch" OR "PLC1_Stop_Active" OR "PLC1_Loi_Tong" THEN
       "V3331_Xa_BonChua1_Man" := FALSE;
   END_IF;
END_REGION

REGION Network 140: Safety override - Reset V3332_Xa_BonChua1
   RUNG wire#powerrail
      Contact( "PLC1_EStop_Latch" )
      wire#w1
      R_Coil( "V3332_Xa_BonChua1" )
   END_RUNG
   RUNG wire#powerrail
      Contact( "PLC1_Stop_Active" )
   END_RUNG wire#w1
   RUNG wire#powerrail
      Contact( "PLC1_Loi_Tong" )
   END_RUNG wire#w1
   // the same network as SCL:
   IF "PLC1_EStop_Latch" OR "PLC1_Stop_Active" OR "PLC1_Loi_Tong" THEN "V3332_Xa_BonChua1" := FALSE; END_IF;
END_REGION

REGION Network 141: Safety override - Reset V3332_Xa_BonChua1_Man
   RUNG wire#powerrail
      Contact( "PLC1_EStop_Latch" )
      wire#w1
      R_Coil( "V3332_Xa_BonChua1_Man" )
   END_RUNG
   RUNG wire#powerrail
      Contact( "PLC1_Stop_Active" )
   END_RUNG wire#w1
   RUNG wire#powerrail
      Contact( "PLC1_Loi_Tong" )
   END_RUNG wire#w1
   // the same network as SCL:
   IF "PLC1_EStop_Latch" OR "PLC1_Stop_Active" OR "PLC1_Loi_Tong" THEN
       "V3332_Xa_BonChua1_Man" := FALSE;
   END_IF;
END_REGION

REGION Network 142: Safety override - Reset V3333_DieuHuong_BonChua1
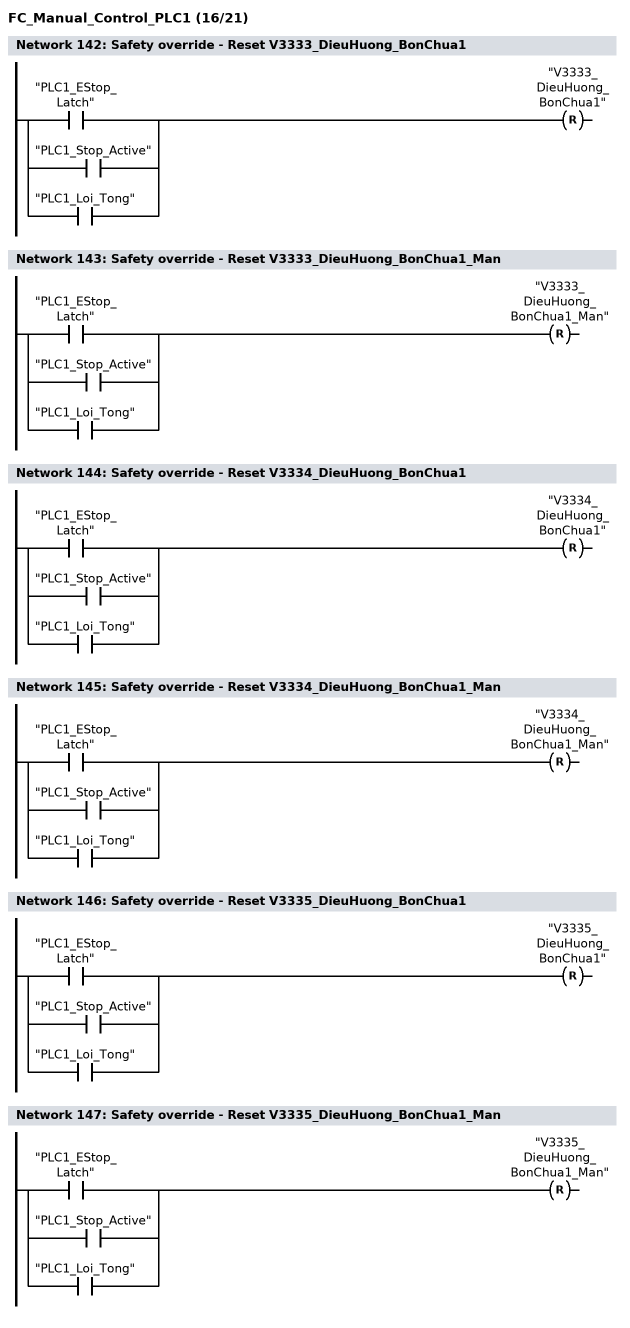
   RUNG wire#powerrail
      Contact( "PLC1_EStop_Latch" )
      wire#w1
      R_Coil( "V3333_DieuHuong_BonChua1" )
   END_RUNG
   RUNG wire#powerrail
      Contact( "PLC1_Stop_Active" )
   END_RUNG wire#w1
   RUNG wire#powerrail
      Contact( "PLC1_Loi_Tong" )
   END_RUNG wire#w1
   // the same network as SCL:
   IF "PLC1_EStop_Latch" OR "PLC1_Stop_Active" OR "PLC1_Loi_Tong" THEN
       "V3333_DieuHuong_BonChua1" := FALSE;
   END_IF;
END_REGION

REGION Network 143: Safety override - Reset V3333_DieuHuong_BonChua1_Man
   RUNG wire#powerrail
      Contact( "PLC1_EStop_Latch" )
      wire#w1
      R_Coil( "V3333_DieuHuong_BonChua1_Man" )
   END_RUNG
   RUNG wire#powerrail
      Contact( "PLC1_Stop_Active" )
   END_RUNG wire#w1
   RUNG wire#powerrail
      Contact( "PLC1_Loi_Tong" )
   END_RUNG wire#w1
   // the same network as SCL:
   IF "PLC1_EStop_Latch" OR "PLC1_Stop_Active" OR "PLC1_Loi_Tong" THEN
       "V3333_DieuHuong_BonChua1_Man" := FALSE;
   END_IF;
END_REGION

REGION Network 144: Safety override - Reset V3334_DieuHuong_BonChua1
   RUNG wire#powerrail
      Contact( "PLC1_EStop_Latch" )
      wire#w1
      R_Coil( "V3334_DieuHuong_BonChua1" )
   END_RUNG
   RUNG wire#powerrail
      Contact( "PLC1_Stop_Active" )
   END_RUNG wire#w1
   RUNG wire#powerrail
      Contact( "PLC1_Loi_Tong" )
   END_RUNG wire#w1
   // the same network as SCL:
   IF "PLC1_EStop_Latch" OR "PLC1_Stop_Active" OR "PLC1_Loi_Tong" THEN
       "V3334_DieuHuong_BonChua1" := FALSE;
   END_IF;
END_REGION

REGION Network 145: Safety override - Reset V3334_DieuHuong_BonChua1_Man
   RUNG wire#powerrail
      Contact( "PLC1_EStop_Latch" )
      wire#w1
      R_Coil( "V3334_DieuHuong_BonChua1_Man" )
   END_RUNG
   RUNG wire#powerrail
      Contact( "PLC1_Stop_Active" )
   END_RUNG wire#w1
   RUNG wire#powerrail
      Contact( "PLC1_Loi_Tong" )
   END_RUNG wire#w1
   // the same network as SCL:
   IF "PLC1_EStop_Latch" OR "PLC1_Stop_Active" OR "PLC1_Loi_Tong" THEN
       "V3334_DieuHuong_BonChua1_Man" := FALSE;
   END_IF;
END_REGION

REGION Network 146: Safety override - Reset V3335_DieuHuong_BonChua1
   RUNG wire#powerrail
      Contact( "PLC1_EStop_Latch" )
      wire#w1
      R_Coil( "V3335_DieuHuong_BonChua1" )
   END_RUNG
   RUNG wire#powerrail
      Contact( "PLC1_Stop_Active" )
   END_RUNG wire#w1
   RUNG wire#powerrail
      Contact( "PLC1_Loi_Tong" )
   END_RUNG wire#w1
   // the same network as SCL:
   IF "PLC1_EStop_Latch" OR "PLC1_Stop_Active" OR "PLC1_Loi_Tong" THEN
       "V3335_DieuHuong_BonChua1" := FALSE;
   END_IF;
END_REGION

REGION Network 147: Safety override - Reset V3335_DieuHuong_BonChua1_Man
   RUNG wire#powerrail
      Contact( "PLC1_EStop_Latch" )
      wire#w1
      R_Coil( "V3335_DieuHuong_BonChua1_Man" )
   END_RUNG
   RUNG wire#powerrail
      Contact( "PLC1_Stop_Active" )
   END_RUNG wire#w1
   RUNG wire#powerrail
      Contact( "PLC1_Loi_Tong" )
   END_RUNG wire#w1
   // the same network as SCL:
   IF "PLC1_EStop_Latch" OR "PLC1_Stop_Active" OR "PLC1_Loi_Tong" THEN
       "V3335_DieuHuong_BonChua1_Man" := FALSE;
   END_IF;
END_REGION

REGION Network 148: Safety override - Reset V3338_Xa_BonChua2
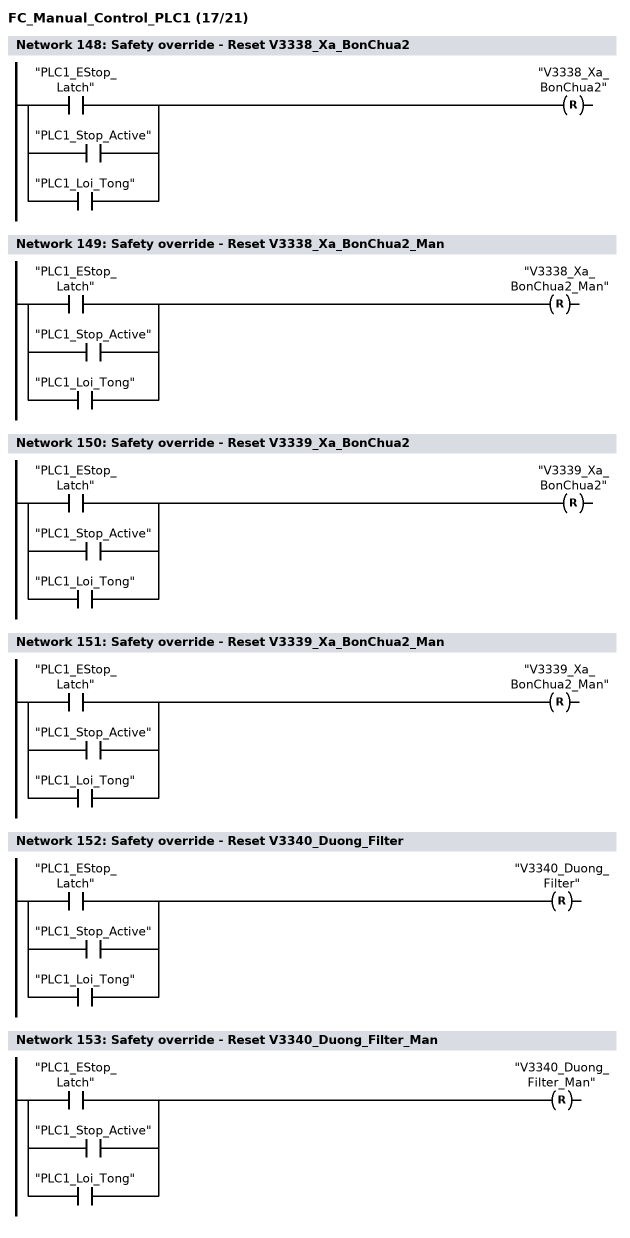
   RUNG wire#powerrail
      Contact( "PLC1_EStop_Latch" )
      wire#w1
      R_Coil( "V3338_Xa_BonChua2" )
   END_RUNG
   RUNG wire#powerrail
      Contact( "PLC1_Stop_Active" )
   END_RUNG wire#w1
   RUNG wire#powerrail
      Contact( "PLC1_Loi_Tong" )
   END_RUNG wire#w1
   // the same network as SCL:
   IF "PLC1_EStop_Latch" OR "PLC1_Stop_Active" OR "PLC1_Loi_Tong" THEN "V3338_Xa_BonChua2" := FALSE; END_IF;
END_REGION

REGION Network 149: Safety override - Reset V3338_Xa_BonChua2_Man
   RUNG wire#powerrail
      Contact( "PLC1_EStop_Latch" )
      wire#w1
      R_Coil( "V3338_Xa_BonChua2_Man" )
   END_RUNG
   RUNG wire#powerrail
      Contact( "PLC1_Stop_Active" )
   END_RUNG wire#w1
   RUNG wire#powerrail
      Contact( "PLC1_Loi_Tong" )
   END_RUNG wire#w1
   // the same network as SCL:
   IF "PLC1_EStop_Latch" OR "PLC1_Stop_Active" OR "PLC1_Loi_Tong" THEN
       "V3338_Xa_BonChua2_Man" := FALSE;
   END_IF;
END_REGION

REGION Network 150: Safety override - Reset V3339_Xa_BonChua2
   RUNG wire#powerrail
      Contact( "PLC1_EStop_Latch" )
      wire#w1
      R_Coil( "V3339_Xa_BonChua2" )
   END_RUNG
   RUNG wire#powerrail
      Contact( "PLC1_Stop_Active" )
   END_RUNG wire#w1
   RUNG wire#powerrail
      Contact( "PLC1_Loi_Tong" )
   END_RUNG wire#w1
   // the same network as SCL:
   IF "PLC1_EStop_Latch" OR "PLC1_Stop_Active" OR "PLC1_Loi_Tong" THEN "V3339_Xa_BonChua2" := FALSE; END_IF;
END_REGION

REGION Network 151: Safety override - Reset V3339_Xa_BonChua2_Man
   RUNG wire#powerrail
      Contact( "PLC1_EStop_Latch" )
      wire#w1
      R_Coil( "V3339_Xa_BonChua2_Man" )
   END_RUNG
   RUNG wire#powerrail
      Contact( "PLC1_Stop_Active" )
   END_RUNG wire#w1
   RUNG wire#powerrail
      Contact( "PLC1_Loi_Tong" )
   END_RUNG wire#w1
   // the same network as SCL:
   IF "PLC1_EStop_Latch" OR "PLC1_Stop_Active" OR "PLC1_Loi_Tong" THEN
       "V3339_Xa_BonChua2_Man" := FALSE;
   END_IF;
END_REGION

REGION Network 152: Safety override - Reset V3340_Duong_Filter
   RUNG wire#powerrail
      Contact( "PLC1_EStop_Latch" )
      wire#w1
      R_Coil( "V3340_Duong_Filter" )
   END_RUNG
   RUNG wire#powerrail
      Contact( "PLC1_Stop_Active" )
   END_RUNG wire#w1
   RUNG wire#powerrail
      Contact( "PLC1_Loi_Tong" )
   END_RUNG wire#w1
   // the same network as SCL:
   IF "PLC1_EStop_Latch" OR "PLC1_Stop_Active" OR "PLC1_Loi_Tong" THEN "V3340_Duong_Filter" := FALSE; END_IF;
END_REGION

REGION Network 153: Safety override - Reset V3340_Duong_Filter_Man
   RUNG wire#powerrail
      Contact( "PLC1_EStop_Latch" )
      wire#w1
      R_Coil( "V3340_Duong_Filter_Man" )
   END_RUNG
   RUNG wire#powerrail
      Contact( "PLC1_Stop_Active" )
   END_RUNG wire#w1
   RUNG wire#powerrail
      Contact( "PLC1_Loi_Tong" )
   END_RUNG wire#w1
   // the same network as SCL:
   IF "PLC1_EStop_Latch" OR "PLC1_Stop_Active" OR "PLC1_Loi_Tong" THEN
       "V3340_Duong_Filter_Man" := FALSE;
   END_IF;
END_REGION

REGION Network 154: Safety override - Reset V3341_Duong_Filter
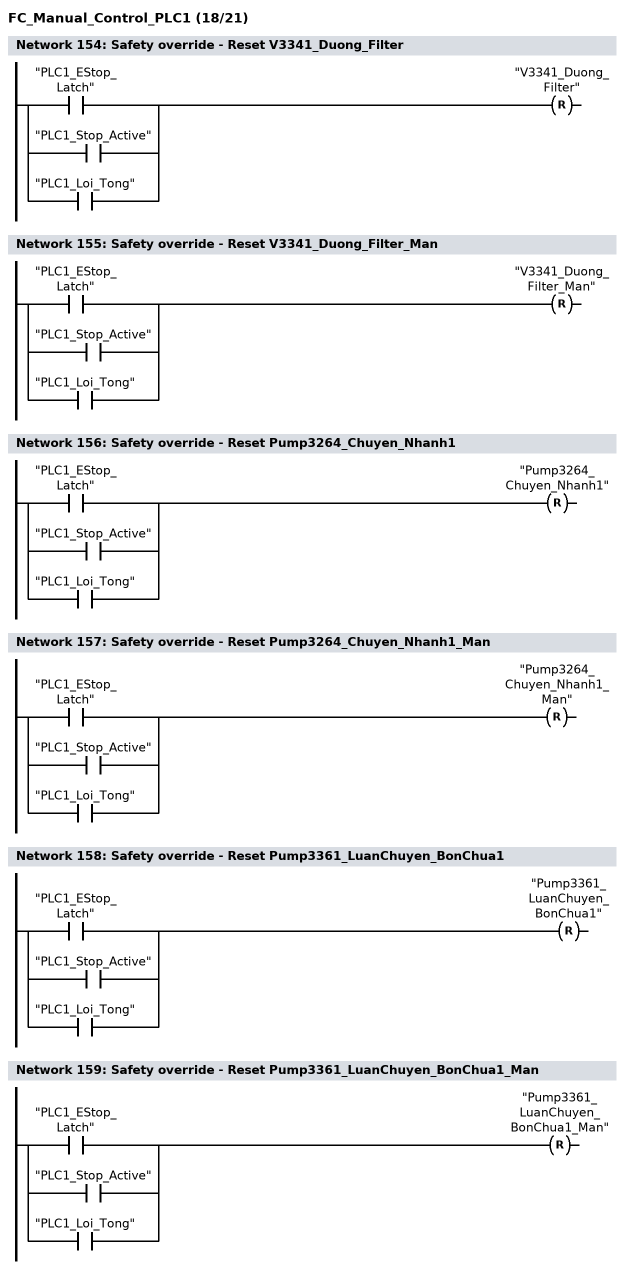
   RUNG wire#powerrail
      Contact( "PLC1_EStop_Latch" )
      wire#w1
      R_Coil( "V3341_Duong_Filter" )
   END_RUNG
   RUNG wire#powerrail
      Contact( "PLC1_Stop_Active" )
   END_RUNG wire#w1
   RUNG wire#powerrail
      Contact( "PLC1_Loi_Tong" )
   END_RUNG wire#w1
   // the same network as SCL:
   IF "PLC1_EStop_Latch" OR "PLC1_Stop_Active" OR "PLC1_Loi_Tong" THEN "V3341_Duong_Filter" := FALSE; END_IF;
END_REGION

REGION Network 155: Safety override - Reset V3341_Duong_Filter_Man
   RUNG wire#powerrail
      Contact( "PLC1_EStop_Latch" )
      wire#w1
      R_Coil( "V3341_Duong_Filter_Man" )
   END_RUNG
   RUNG wire#powerrail
      Contact( "PLC1_Stop_Active" )
   END_RUNG wire#w1
   RUNG wire#powerrail
      Contact( "PLC1_Loi_Tong" )
   END_RUNG wire#w1
   // the same network as SCL:
   IF "PLC1_EStop_Latch" OR "PLC1_Stop_Active" OR "PLC1_Loi_Tong" THEN
       "V3341_Duong_Filter_Man" := FALSE;
   END_IF;
END_REGION

REGION Network 156: Safety override - Reset Pump3264_Chuyen_Nhanh1
   RUNG wire#powerrail
      Contact( "PLC1_EStop_Latch" )
      wire#w1
      R_Coil( "Pump3264_Chuyen_Nhanh1" )
   END_RUNG
   RUNG wire#powerrail
      Contact( "PLC1_Stop_Active" )
   END_RUNG wire#w1
   RUNG wire#powerrail
      Contact( "PLC1_Loi_Tong" )
   END_RUNG wire#w1
   // the same network as SCL:
   IF "PLC1_EStop_Latch" OR "PLC1_Stop_Active" OR "PLC1_Loi_Tong" THEN
       "Pump3264_Chuyen_Nhanh1" := FALSE;
   END_IF;
END_REGION

REGION Network 157: Safety override - Reset Pump3264_Chuyen_Nhanh1_Man
   RUNG wire#powerrail
      Contact( "PLC1_EStop_Latch" )
      wire#w1
      R_Coil( "Pump3264_Chuyen_Nhanh1_Man" )
   END_RUNG
   RUNG wire#powerrail
      Contact( "PLC1_Stop_Active" )
   END_RUNG wire#w1
   RUNG wire#powerrail
      Contact( "PLC1_Loi_Tong" )
   END_RUNG wire#w1
   // the same network as SCL:
   IF "PLC1_EStop_Latch" OR "PLC1_Stop_Active" OR "PLC1_Loi_Tong" THEN
       "Pump3264_Chuyen_Nhanh1_Man" := FALSE;
   END_IF;
END_REGION

REGION Network 158: Safety override - Reset Pump3361_LuanChuyen_BonChua1
   RUNG wire#powerrail
      Contact( "PLC1_EStop_Latch" )
      wire#w1
      R_Coil( "Pump3361_LuanChuyen_BonChua1" )
   END_RUNG
   RUNG wire#powerrail
      Contact( "PLC1_Stop_Active" )
   END_RUNG wire#w1
   RUNG wire#powerrail
      Contact( "PLC1_Loi_Tong" )
   END_RUNG wire#w1
   // the same network as SCL:
   IF "PLC1_EStop_Latch" OR "PLC1_Stop_Active" OR "PLC1_Loi_Tong" THEN
       "Pump3361_LuanChuyen_BonChua1" := FALSE;
   END_IF;
END_REGION

REGION Network 159: Safety override - Reset Pump3361_LuanChuyen_BonChua1_Man
   RUNG wire#powerrail
      Contact( "PLC1_EStop_Latch" )
      wire#w1
      R_Coil( "Pump3361_LuanChuyen_BonChua1_Man" )
   END_RUNG
   RUNG wire#powerrail
      Contact( "PLC1_Stop_Active" )
   END_RUNG wire#w1
   RUNG wire#powerrail
      Contact( "PLC1_Loi_Tong" )
   END_RUNG wire#w1
   // the same network as SCL:
   IF "PLC1_EStop_Latch" OR "PLC1_Stop_Active" OR "PLC1_Loi_Tong" THEN
       "Pump3361_LuanChuyen_BonChua1_Man" := FALSE;
   END_IF;
END_REGION

REGION Network 160: Safety override - Reset Pump3362_Xa_BonChua1
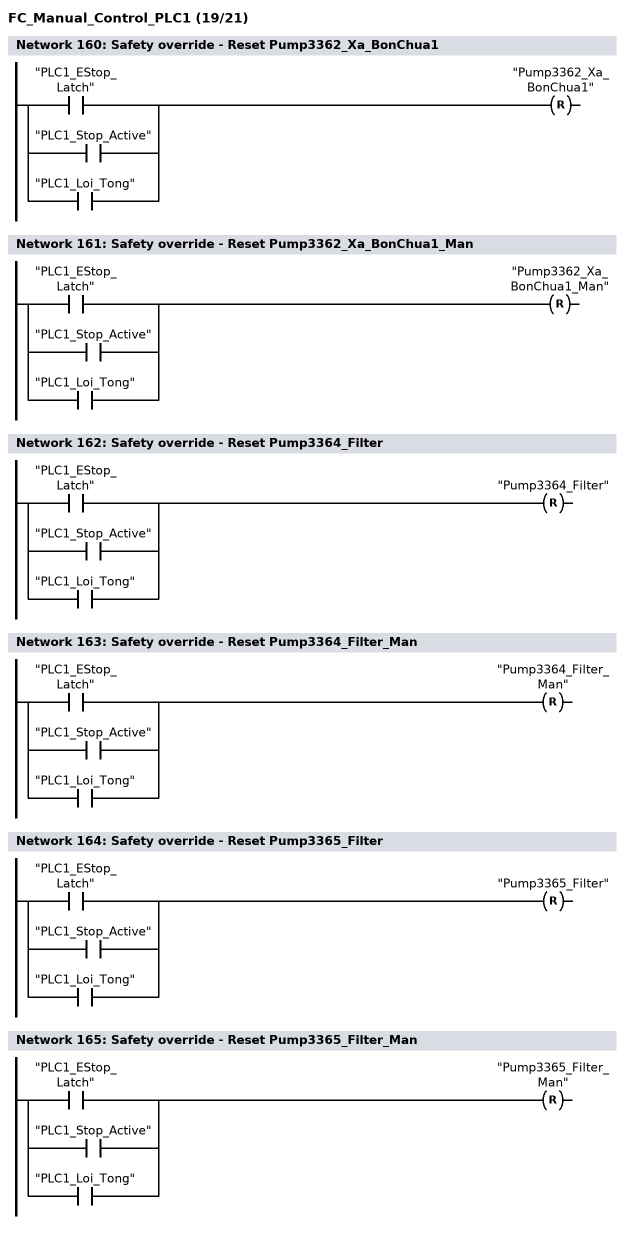
   RUNG wire#powerrail
      Contact( "PLC1_EStop_Latch" )
      wire#w1
      R_Coil( "Pump3362_Xa_BonChua1" )
   END_RUNG
   RUNG wire#powerrail
      Contact( "PLC1_Stop_Active" )
   END_RUNG wire#w1
   RUNG wire#powerrail
      Contact( "PLC1_Loi_Tong" )
   END_RUNG wire#w1
   // the same network as SCL:
   IF "PLC1_EStop_Latch" OR "PLC1_Stop_Active" OR "PLC1_Loi_Tong" THEN
       "Pump3362_Xa_BonChua1" := FALSE;
   END_IF;
END_REGION

REGION Network 161: Safety override - Reset Pump3362_Xa_BonChua1_Man
   RUNG wire#powerrail
      Contact( "PLC1_EStop_Latch" )
      wire#w1
      R_Coil( "Pump3362_Xa_BonChua1_Man" )
   END_RUNG
   RUNG wire#powerrail
      Contact( "PLC1_Stop_Active" )
   END_RUNG wire#w1
   RUNG wire#powerrail
      Contact( "PLC1_Loi_Tong" )
   END_RUNG wire#w1
   // the same network as SCL:
   IF "PLC1_EStop_Latch" OR "PLC1_Stop_Active" OR "PLC1_Loi_Tong" THEN
       "Pump3362_Xa_BonChua1_Man" := FALSE;
   END_IF;
END_REGION

REGION Network 162: Safety override - Reset Pump3364_Filter
   RUNG wire#powerrail
      Contact( "PLC1_EStop_Latch" )
      wire#w1
      R_Coil( "Pump3364_Filter" )
   END_RUNG
   RUNG wire#powerrail
      Contact( "PLC1_Stop_Active" )
   END_RUNG wire#w1
   RUNG wire#powerrail
      Contact( "PLC1_Loi_Tong" )
   END_RUNG wire#w1
   // the same network as SCL:
   IF "PLC1_EStop_Latch" OR "PLC1_Stop_Active" OR "PLC1_Loi_Tong" THEN "Pump3364_Filter" := FALSE; END_IF;
END_REGION

REGION Network 163: Safety override - Reset Pump3364_Filter_Man
   RUNG wire#powerrail
      Contact( "PLC1_EStop_Latch" )
      wire#w1
      R_Coil( "Pump3364_Filter_Man" )
   END_RUNG
   RUNG wire#powerrail
      Contact( "PLC1_Stop_Active" )
   END_RUNG wire#w1
   RUNG wire#powerrail
      Contact( "PLC1_Loi_Tong" )
   END_RUNG wire#w1
   // the same network as SCL:
   IF "PLC1_EStop_Latch" OR "PLC1_Stop_Active" OR "PLC1_Loi_Tong" THEN
       "Pump3364_Filter_Man" := FALSE;
   END_IF;
END_REGION

REGION Network 164: Safety override - Reset Pump3365_Filter
   RUNG wire#powerrail
      Contact( "PLC1_EStop_Latch" )
      wire#w1
      R_Coil( "Pump3365_Filter" )
   END_RUNG
   RUNG wire#powerrail
      Contact( "PLC1_Stop_Active" )
   END_RUNG wire#w1
   RUNG wire#powerrail
      Contact( "PLC1_Loi_Tong" )
   END_RUNG wire#w1
   // the same network as SCL:
   IF "PLC1_EStop_Latch" OR "PLC1_Stop_Active" OR "PLC1_Loi_Tong" THEN "Pump3365_Filter" := FALSE; END_IF;
END_REGION

REGION Network 165: Safety override - Reset Pump3365_Filter_Man
   RUNG wire#powerrail
      Contact( "PLC1_EStop_Latch" )
      wire#w1
      R_Coil( "Pump3365_Filter_Man" )
   END_RUNG
   RUNG wire#powerrail
      Contact( "PLC1_Stop_Active" )
   END_RUNG wire#w1
   RUNG wire#powerrail
      Contact( "PLC1_Loi_Tong" )
   END_RUNG wire#w1
   // the same network as SCL:
   IF "PLC1_EStop_Latch" OR "PLC1_Stop_Active" OR "PLC1_Loi_Tong" THEN
       "Pump3365_Filter_Man" := FALSE;
   END_IF;
END_REGION

REGION Network 166: Safety override - Clear CV3201_Nuoc_Bon1
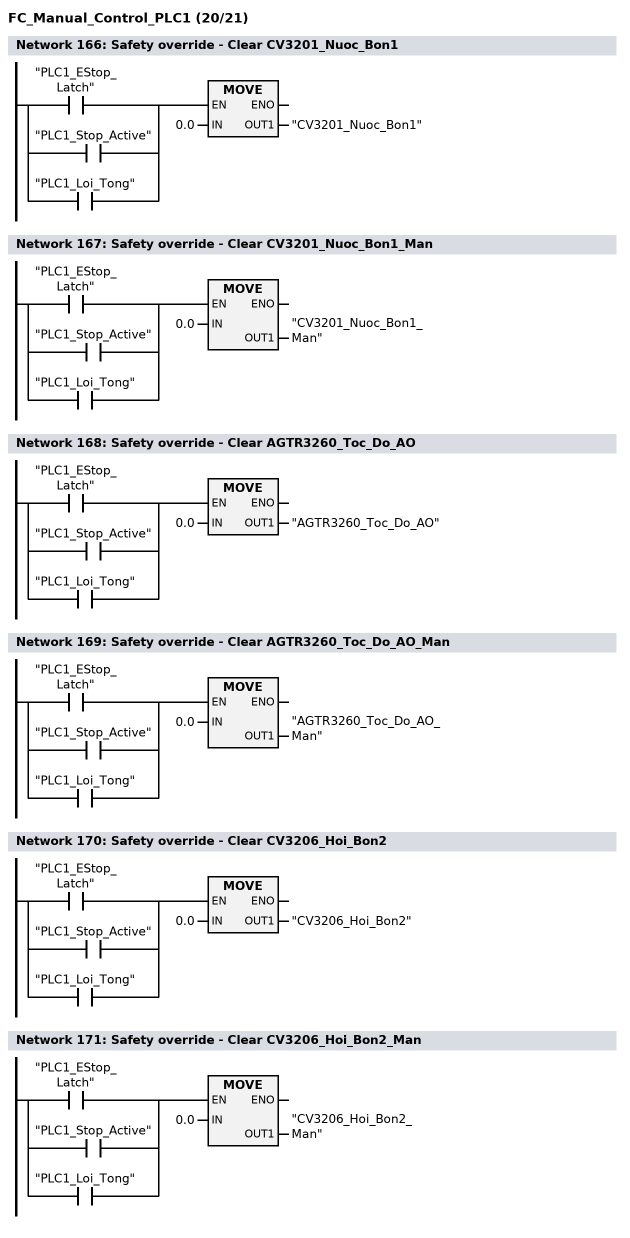
   RUNG wire#powerrail
      Contact( "PLC1_EStop_Latch" )
      wire#w1
      { S7_GenerateENO := "TRUE" } Move(in := 0.0, out1 => "CV3201_Nuoc_Bon1")
   END_RUNG
   RUNG wire#powerrail
      Contact( "PLC1_Stop_Active" )
   END_RUNG wire#w1
   RUNG wire#powerrail
      Contact( "PLC1_Loi_Tong" )
   END_RUNG wire#w1
   // the same network as SCL:
   IF "PLC1_EStop_Latch" OR "PLC1_Stop_Active" OR "PLC1_Loi_Tong" THEN "CV3201_Nuoc_Bon1" := 0.0; END_IF;
END_REGION

REGION Network 167: Safety override - Clear CV3201_Nuoc_Bon1_Man
   RUNG wire#powerrail
      Contact( "PLC1_EStop_Latch" )
      wire#w1
      { S7_GenerateENO := "TRUE" } Move(in := 0.0, out1 => "CV3201_Nuoc_Bon1_Man")
   END_RUNG
   RUNG wire#powerrail
      Contact( "PLC1_Stop_Active" )
   END_RUNG wire#w1
   RUNG wire#powerrail
      Contact( "PLC1_Loi_Tong" )
   END_RUNG wire#w1
   // the same network as SCL:
   IF "PLC1_EStop_Latch" OR "PLC1_Stop_Active" OR "PLC1_Loi_Tong" THEN "CV3201_Nuoc_Bon1_Man" := 0.0; END_IF;
END_REGION

REGION Network 168: Safety override - Clear AGTR3260_Toc_Do_AO
   RUNG wire#powerrail
      Contact( "PLC1_EStop_Latch" )
      wire#w1
      { S7_GenerateENO := "TRUE" } Move(in := 0.0, out1 => "AGTR3260_Toc_Do_AO")
   END_RUNG
   RUNG wire#powerrail
      Contact( "PLC1_Stop_Active" )
   END_RUNG wire#w1
   RUNG wire#powerrail
      Contact( "PLC1_Loi_Tong" )
   END_RUNG wire#w1
   // the same network as SCL:
   IF "PLC1_EStop_Latch" OR "PLC1_Stop_Active" OR "PLC1_Loi_Tong" THEN "AGTR3260_Toc_Do_AO" := 0.0; END_IF;
END_REGION

REGION Network 169: Safety override - Clear AGTR3260_Toc_Do_AO_Man
   RUNG wire#powerrail
      Contact( "PLC1_EStop_Latch" )
      wire#w1
      { S7_GenerateENO := "TRUE" } Move(in := 0.0, out1 => "AGTR3260_Toc_Do_AO_Man")
   END_RUNG
   RUNG wire#powerrail
      Contact( "PLC1_Stop_Active" )
   END_RUNG wire#w1
   RUNG wire#powerrail
      Contact( "PLC1_Loi_Tong" )
   END_RUNG wire#w1
   // the same network as SCL:
   IF "PLC1_EStop_Latch" OR "PLC1_Stop_Active" OR "PLC1_Loi_Tong" THEN
       "AGTR3260_Toc_Do_AO_Man" := 0.0;
   END_IF;
END_REGION

REGION Network 170: Safety override - Clear CV3206_Hoi_Bon2
   RUNG wire#powerrail
      Contact( "PLC1_EStop_Latch" )
      wire#w1
      { S7_GenerateENO := "TRUE" } Move(in := 0.0, out1 => "CV3206_Hoi_Bon2")
   END_RUNG
   RUNG wire#powerrail
      Contact( "PLC1_Stop_Active" )
   END_RUNG wire#w1
   RUNG wire#powerrail
      Contact( "PLC1_Loi_Tong" )
   END_RUNG wire#w1
   // the same network as SCL:
   IF "PLC1_EStop_Latch" OR "PLC1_Stop_Active" OR "PLC1_Loi_Tong" THEN "CV3206_Hoi_Bon2" := 0.0; END_IF;
END_REGION

REGION Network 171: Safety override - Clear CV3206_Hoi_Bon2_Man
   RUNG wire#powerrail
      Contact( "PLC1_EStop_Latch" )
      wire#w1
      { S7_GenerateENO := "TRUE" } Move(in := 0.0, out1 => "CV3206_Hoi_Bon2_Man")
   END_RUNG
   RUNG wire#powerrail
      Contact( "PLC1_Stop_Active" )
   END_RUNG wire#w1
   RUNG wire#powerrail
      Contact( "PLC1_Loi_Tong" )
   END_RUNG wire#w1
   // the same network as SCL:
   IF "PLC1_EStop_Latch" OR "PLC1_Stop_Active" OR "PLC1_Loi_Tong" THEN "CV3206_Hoi_Bon2_Man" := 0.0; END_IF;
END_REGION

REGION Network 172: Safety override - Clear VFD_Bon2_Toc_Do_Cmd
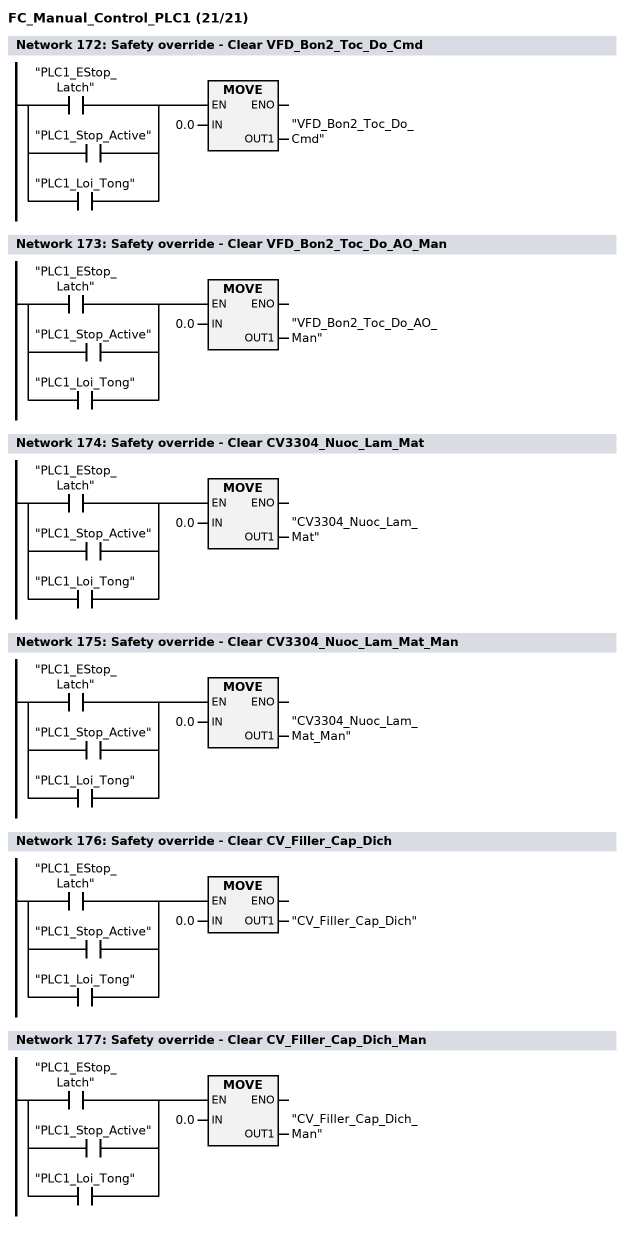
   RUNG wire#powerrail
      Contact( "PLC1_EStop_Latch" )
      wire#w1
      { S7_GenerateENO := "TRUE" } Move(in := 0.0, out1 => "VFD_Bon2_Toc_Do_Cmd")
   END_RUNG
   RUNG wire#powerrail
      Contact( "PLC1_Stop_Active" )
   END_RUNG wire#w1
   RUNG wire#powerrail
      Contact( "PLC1_Loi_Tong" )
   END_RUNG wire#w1
   // the same network as SCL:
   IF "PLC1_EStop_Latch" OR "PLC1_Stop_Active" OR "PLC1_Loi_Tong" THEN "VFD_Bon2_Toc_Do_Cmd" := 0.0; END_IF;
END_REGION

REGION Network 173: Safety override - Clear VFD_Bon2_Toc_Do_AO_Man
   RUNG wire#powerrail
      Contact( "PLC1_EStop_Latch" )
      wire#w1
      { S7_GenerateENO := "TRUE" } Move(in := 0.0, out1 => "VFD_Bon2_Toc_Do_AO_Man")
   END_RUNG
   RUNG wire#powerrail
      Contact( "PLC1_Stop_Active" )
   END_RUNG wire#w1
   RUNG wire#powerrail
      Contact( "PLC1_Loi_Tong" )
   END_RUNG wire#w1
   // the same network as SCL:
   IF "PLC1_EStop_Latch" OR "PLC1_Stop_Active" OR "PLC1_Loi_Tong" THEN
       "VFD_Bon2_Toc_Do_AO_Man" := 0.0;
   END_IF;
END_REGION

REGION Network 174: Safety override - Clear CV3304_Nuoc_Lam_Mat
   RUNG wire#powerrail
      Contact( "PLC1_EStop_Latch" )
      wire#w1
      { S7_GenerateENO := "TRUE" } Move(in := 0.0, out1 => "CV3304_Nuoc_Lam_Mat")
   END_RUNG
   RUNG wire#powerrail
      Contact( "PLC1_Stop_Active" )
   END_RUNG wire#w1
   RUNG wire#powerrail
      Contact( "PLC1_Loi_Tong" )
   END_RUNG wire#w1
   // the same network as SCL:
   IF "PLC1_EStop_Latch" OR "PLC1_Stop_Active" OR "PLC1_Loi_Tong" THEN "CV3304_Nuoc_Lam_Mat" := 0.0; END_IF;
END_REGION

REGION Network 175: Safety override - Clear CV3304_Nuoc_Lam_Mat_Man
   RUNG wire#powerrail
      Contact( "PLC1_EStop_Latch" )
      wire#w1
      { S7_GenerateENO := "TRUE" } Move(in := 0.0, out1 => "CV3304_Nuoc_Lam_Mat_Man")
   END_RUNG
   RUNG wire#powerrail
      Contact( "PLC1_Stop_Active" )
   END_RUNG wire#w1
   RUNG wire#powerrail
      Contact( "PLC1_Loi_Tong" )
   END_RUNG wire#w1
   // the same network as SCL:
   IF "PLC1_EStop_Latch" OR "PLC1_Stop_Active" OR "PLC1_Loi_Tong" THEN
       "CV3304_Nuoc_Lam_Mat_Man" := 0.0;
   END_IF;
END_REGION

REGION Network 176: Safety override - Clear CV_Filler_Cap_Dich
   RUNG wire#powerrail
      Contact( "PLC1_EStop_Latch" )
      wire#w1
      { S7_GenerateENO := "TRUE" } Move(in := 0.0, out1 => "CV_Filler_Cap_Dich")
   END_RUNG
   RUNG wire#powerrail
      Contact( "PLC1_Stop_Active" )
   END_RUNG wire#w1
   RUNG wire#powerrail
      Contact( "PLC1_Loi_Tong" )
   END_RUNG wire#w1
   // the same network as SCL:
   IF "PLC1_EStop_Latch" OR "PLC1_Stop_Active" OR "PLC1_Loi_Tong" THEN "CV_Filler_Cap_Dich" := 0.0; END_IF;
END_REGION

REGION Network 177: Safety override - Clear CV_Filler_Cap_Dich_Man
   RUNG wire#powerrail
      Contact( "PLC1_EStop_Latch" )
      wire#w1
      { S7_GenerateENO := "TRUE" } Move(in := 0.0, out1 => "CV_Filler_Cap_Dich_Man")
   END_RUNG
   RUNG wire#powerrail
      Contact( "PLC1_Stop_Active" )
   END_RUNG wire#w1
   RUNG wire#powerrail
      Contact( "PLC1_Loi_Tong" )
   END_RUNG wire#w1
   // the same network as SCL:
   IF "PLC1_EStop_Latch" OR "PLC1_Stop_Active" OR "PLC1_Loi_Tong" THEN
       "CV_Filler_Cap_Dich_Man" := 0.0;
   END_IF;
END_REGION
END_FUNCTION
